# B&R Automation Studio project ABC_Pltzr (part 3)

#### paiPVSerDesMgr.typ
```iecst
(********************************************************************
 * COPYRIGHT --
 ********************************************************************
 * Package: paiFileService
 * File: paiPVSerDesMgr
 * Author: goran_2
 * Created: August 05, 2015
 ********************************************************************
 * Data types of package paiFileService
 ********************************************************************)

TYPE
	paiFSEnums_typ :
		(
		PAI_FS_PVNAME_MAXLEN := 63,
		PAI_FS_PATH_MAXLEN := 127,
		PAI_FS_TXTLEN_MID := 127,
		PAI_FS_SERDESMGR_PWRUP_NA := 0, (*PV restore option at Power Up: no action*)
		PAI_FS_SERDESMGR_PWRUP_DFLT := 1, (*PV restore option at Power Up: test storage, if different preload defaults*)
		PAI_FS_SERDESMGR_PWRUP_DFLT_fRD := 2, (*PV restore option at Power Up: test storage, if different preload defaults then read data from file*)
		PAI_FS_SERDESMGR_MAXITEMIDX := 19
		);
	paiPVSerDesChangeMonitor_typ : 	STRUCT  (*Change monitor: optional feature*)
		iChngEnable : BOOL; (*0-disabled;1-enabled*)
		iChngRejected : BOOL; (*1-reject PV changes, restore previous value*)
		iChngAccepted : BOOL; (*1-accept PV changes, store PV to file*)
		oChngDetected : BOOL; (*1-PV is changed, use information to prompt user*)
		oError : UDINT; (*1-option is enabled, but provided memory is unsufficent*)
		oState : UDINT; (*1-option is enabled, but provided memory is unsufficent*)
		iChangeMonitorMemSize : UDINT; (*size of the address space for this feature (shall be the same size or greater than the size of the PV)*)
		pChangeMonitorMem : UDINT; (*ptr to address space which has the same size as the PV (use for memory compare to detect changes)*)
	END_STRUCT;
	paiPVSerDesHMI_typ : 	STRUCT
		iBtnChangeReject : USINT;
		iBtnChangeAccept : USINT;
		iBtnSerRequest : USINT;
		iBtnDesRequest : USINT;
		oBtnVisible : USINT;
		oBtnClick : USINT;
	END_STRUCT;
	paiPVSerDesPowerUp_typ : 	STRUCT  (*Option: control of a behaivor at power up*)
		iPowerUpConfig : UDINT; (*0-nothing to do; 1-use test data; if diff, run defaults; 2-use test data; if diff, read from file*)
		iTestData : UDINT; (*Test data value (i.e. magic word 0x55555555)*)
		pTestDataStorage : UDINT; (*Ptr to the location of the magic word for this variable*)
		oError : UDINT; (*0-not ready after power up; 1-ready after power up*)
		oInitReady : UDINT; (*0-not ready after power up; 1-ready after power up*)
		oStatus : STRING[15]; (*0-not ready after power up; 1-ready after power up*)
	END_STRUCT;
	paiPVSerDesItem_typ : 	STRUCT
		iPVName : STRING[PAI_FS_PVNAME_MAXLEN]; (*PV name*)
		iDevicename : STRING[PAI_FS_PVNAME_MAXLEN]; (*Name of the file device to store PV*)
		iFilename : STRING[PAI_FS_PATH_MAXLEN]; (*Filename to store PV*)
		iSerRequest : BOOL; (*Request to write PV to file (i.e. serialize PV to file buffer > write data to  file)*)
		iDesRequest : BOOL; (*Request to read PV from file (i.e. read file to file buffer > deserialize data to PV)*)
		pPV : UDINT; (*ptr to PV*)
		iPVSize : UDINT; (*size of the PV (in bytes)*)
		pFilebuffer : UDINT; (*ptr to file r/w buffer*)
		iFilebufferSize : UDINT; (*size (bytes) of the file r/w buffer*)
		optChangeMonitor : paiPVSerDesChangeMonitor_typ; (*optional feature for automatic / HMI assisted read/write of PV-s upon changes*)
		optInitAtPowerUp : paiPVSerDesPowerUp_typ; (*optional feature: control PV init at power up; see above*)
		optPtrHMIData : REFERENCE TO paiPVSerDesHMI_typ; (*optional feature: HMI interface for PV read/write to/from file*)
		pCallbackDes : UDINT; (*deserialize callback function - processes PV deser request*)
		pCallbackSer : UDINT; (*serialize callback function - processes PV serialize request*)
		pCallbackDefault : UDINT; (*default callback function - function to set PV default values*)
		oState : UDINT; (*mgr current state*)
		oDone : UDINT; (*1 - ser or deser request is complete; *)
		oSerCount : UDINT;
		oDesCount : UDINT;
		oSerCountOld : UDINT;
		oDesCountOld : UDINT;
		oFilesizeLastSer : UDINT;
		oFilesizeLastDes : UDINT;
		oTimestampLastSer : STRING[63];
		oTimestampLastDes : STRING[63];
		oErrorCount : UDINT;
		oErrorCountOld : UDINT;
		oError : UDINT;
		oErrorTxt : STRING[PAI_FS_TXTLEN_MID];
	END_STRUCT;
	paiPVSerDesMgr_typ : 	STRUCT
		pPaiFS : UDINT;
		oState : UDINT;
		iItemCount : UDINT;
		pvItems : ARRAY[0..PAI_FS_SERDESMGR_MAXITEMIDX]OF paiPVSerDesItem_typ;
	END_STRUCT;
END_TYPE
```

#### paiFileService.var
```iecst
(********************************************************************
 * COPYRIGHT --
 ********************************************************************
 * Package: paiFileService
 * File: paiFileService.var
 * Author: goran_2
 * Created: August 05, 2011
 ********************************************************************
 * Variables of package paiFileService
 ********************************************************************)
VAR
	paiFS : paiFileService_typ := (0); (*Global PV for interfacing to PAI file service.*)
	paiFSDevices : paiFileServiceDeviceTable_typ := (0);
END_VAR
```

#### paiPVSerDesMgr.h
```c
/********************************************************************
 * COPYRIGHT --
 ********************************************************************
 * Package: paiFileService
 * File: paiPVSerDesMgr.h
 * Author: goran
 * Created: August 18, 2015
 *******************************************************************/

#include <bur/plctypes.h>

void paiPVSerDesMgrInit(paiPVSerDesMgr_typ* p);
void paiPVSerDesMgrCyclic(paiPVSerDesMgr_typ* p);

//callback functions
void paiCBWriteFileSerPV(paiFileService_typ* p, UDINT pCallbackData);
void paiCBReadFileDesPV(paiFileService_typ* p, UDINT pCallbackData);

//EOF
```

#### paiFSInterface.c
```c
/********************************************************************
 * COPYRIGHT --
 ********************************************************************
 * Package: paiFileService
 * File: paiFSInterface.c
 * Author: goran
 * Created: August 18, 2015
 *******************************************************************/

#include <bur/plctypes.h>
#ifdef _DEFAULT_INCLUDES
	#include <AsDefault.h>
#endif

#include "paiFSInterface.h"

/*
###############################################################################
Utility function to access paiFS service
###############################################################################
*/
void paiFSSetCallback(paiFileService_typ* p, UDINT pCallback, UDINT pCallbackData)
{
	if(!p)
		return;

	p->i.pCallback = pCallback;
	p->i.pCallbackData = pCallbackData;
}

void paiFSExeCallback(paiFileService_typ* p)
{
	if(!p)
		return;

	//execute fs callback to enable app to process file io
	if(p->i.pCallback){
		void (*fsCB)(paiFileService_typ* pFS, UDINT pCallbackData) =  ( void(*) (paiFileService_typ* pFS, UDINT pCallbackData) ) p->i.pCallback;
		(*fsCB)(p, p->i.pCallbackData);
	}
}

void paiFSExeCallbackCyclic(paiFileService_typ* p)
{
	//wait until request completes
	if( paiFSFileRequestIsBusy(p) )
		return;

	if( p->o.done ){
		//clear done event
		p->o.done = 0;

		//execute call back after file IO command execution is complete
		paiFSExeCallback(p);
	}
}

void paiFSDirCreateRequest(paiFileService_typ* p, UDINT adrDeviceName, UDINT adrPath, UDINT pCallback, UDINT pCallbackData)
{
	p->i.request = PAI_FS_CRDIR;
	p->i.adrName = (UDINT)adrPath;
	p->i.adrDeviceName = (UDINT) adrDeviceName;
	paiFSSetCallback(p, pCallback, pCallbackData);
}

void paiFSDirInfoRequest(paiFileService_typ* p, UDINT adrDeviceName, UDINT adrPath, UDINT pCallback, UDINT pCallbackData)
{
	p->i.request = PAI_FS_INFODIR;
	p->i.adrName = (UDINT)adrPath;
	p->i.adrDeviceName = (UDINT) adrDeviceName;
	paiFSSetCallback(p, pCallback, pCallbackData);
}

void paiFSFileDelRequest(paiFileService_typ* p, UDINT adrDeviceName, UDINT adrName, UDINT pCallback, UDINT pCallbackData)
{
	p->i.request = PAI_FS_DELFILE;
	p->i.adrName = (UDINT)adrName;
	p->i.adrDeviceName = (UDINT) adrDeviceName;
	paiFSSetCallback(p, pCallback, pCallbackData);
}

void paiFSFileRdRequest(paiFileService_typ* p, UDINT adrDeviceName, UDINT adrName, UDINT adrDst, UDINT sizeDst, UDINT pCallback, UDINT pCallbackData)
{
	p->i.request = PAI_FS_RDFILE;
	p->i.adrDeviceName = (UDINT) adrDeviceName;
	p->i.adrName = (UDINT)adrName;
	p->i.adrReadDst = (UDINT)adrDst;
	p->i.readDstLen = sizeDst;
	paiFSSetCallback(p, pCallback, pCallbackData);
}

void paiFSFileWrRequest(paiFileService_typ* p, UDINT adrDeviceName, UDINT adrName, UDINT adrSrc, UDINT sizeSrc, UDINT pCallback, UDINT pCallbackData)
{
	p->i.request= PAI_FS_WRFILE;
	p->i.adrDeviceName = (UDINT) adrDeviceName;
	p->i.adrName = (UDINT)adrName;
	p->i.adrWriteSrc = (UDINT)adrSrc;
	p->i.writeSrcLen= sizeSrc;
	paiFSSetCallback(p, pCallback, pCallbackData);
}

BOOL paiFSFileRequestIsBusy(paiFileService_typ* p)
{
	//wait until request completes
	if(p->o.busy)
		return 1;

	//reset request! IMPORTANT!
	p->i.request = PAI_FS_IDLE;
	return 0;
}

BOOL paiFSFileSystemIsInit(paiFileService_typ* p)
{
	if(!p->o.initOk)	//can't do much before paiFS completes
		return 0;

	return 1;
}
```

#### Program Logical/paiComponents/paiFileService/paiFSUnitTest

##### paiFSUnitTest.c
```c
/********************************************************************
 * COPYRIGHT --
 ********************************************************************
 * Program: paiFileTestClient
 * File: paiFileTestClient.c
 * Author: goran_2
 * Created: August 05, 2011
 ********************************************************************
 * Implementation of program paiFileTestClient
 ********************************************************************/

#include <bur/plctypes.h>

#ifdef _DEFAULT_INCLUDES
 #include <AsDefault.h>
#endif

/*
###############################################################################
PV-s
###############################################################################
*/

/*
###############################################################################
PV-s
###############################################################################
*/
#define BUF_LEN 1000
_LOCAL char txt[BUF_LEN];

_LOCAL char filename[32];

_LOCAL int readcounterok ;
_LOCAL int readcountererr ;

_LOCAL int writecounterok ;
_LOCAL int writecountererr ;

_LOCAL int myInitDone;

/*
###############################################################################
Init, Cyclic, Exit
###############################################################################
*/
void _INIT paiFileTestClientINIT( void )
{
	/* TODO: Add code here */
	myInitDone = 0;
}

void _CYCLIC paiFileTestClientCYCLIC( void )
{
	/* TODO: Add code here */

	/*wait till file service ready then init application access to file service*/
	if(!myInitDone && paiFS.io.initOk){
		myInitDone = 1;
		/*copy filename into a buffer so it may be changed from the watch window*/
		strcpy(filename, "appcfg.txt");
		paiFS.io.fileName = (UDINT)filename;

		/*in this example same buffer used for read and write*/
		paiFS.io.readDstAdr = (UDINT)txt;
		paiFS.io.readDstLen = BUF_LEN;
		paiFS.io.writeSrcAdr= (UDINT)txt;

		/*aux PV-s to monitor the activity*/
		readcounterok = 0;
		readcountererr = 0;

		writecounterok = 0;
		writecountererr = 0;
	}

	/*in this example continously update length for write request. That way, when writeRequest get's issued from watch window, correct value gets set!*/
	paiFS.io.writeSrcLen = strlen(&txt[0]);

	/*example on how to monitor if file service has completed a request*/
	if(paiFS.io.readDone){
		/*reset signal here*/
		paiFS.io.readDone = 0;

		if(paiFS.io.status)
			readcountererr++;
		else
			readcounterok++;
	}

	if(paiFS.io.writeDone){
		/*reset signal here*/
		paiFS.io.writeDone = 0;

		if(paiFS.io.status)
			writecountererr++;
		else
			writecounterok++;
	}
}

void _EXIT paiFileTestClientEXIT( void )
{
	/* TODO: Add code here */
}
```

### Program Logical/paiComponents/paiHmi

#### paiHmiCmd.typ
```iecst
(********************************************************************
 * COPYRIGHT -- pai
 ********************************************************************
 * Package: HMI
 * File: HMI.typ
 * Author: goran
 * Created: August 28, 2013
 ********************************************************************
 * Data types of package HMI
 ********************************************************************)
(*==========================*)
(*==== HMI Command Interface ==*)
(*==========================*)

TYPE
	hmiCmd_typ : 	STRUCT
		main : hmiCmdMain_typ;
		infeed : hmiCmdInfeed_typ;
		outfeed : hmiCmdOutfeed_typ;
		qc : hmiCmdQC_typ;
		lights : hmiCmdLights_typ;
		diag : hmiCmdDiag_typ;
		listQCInspectors : STRING[511];
	END_STRUCT;
	hmiCmdX20Outfeed_typ : 	STRUCT  (*command to control / force an OUTFEED output module*)
		doDoorWeigh : BOOL; (*weigh door*)
		doBelt : BOOL; (*belt control clutch*)
		doQC1 : BOOL; (*qc1 diverter *)
		doQC2 : BOOL; (*qc2 diverter*)
	END_STRUCT;
	hmiCmdX20Station_typ : 	STRUCT  (*command to control / force an STATION output module(s)*)
		doTakeout0 : BOOL; (*takeout (0 + moduleNum*4)*)
		doTakeout1 : BOOL; (*takeout (1 + moduleNum*4)*)
		doTakeout2 : BOOL; (*takeout (2 + moduleNum*4)*)
		doTakeout3 : BOOL; (*takeout (3 + moduleNum*4)*)
		doDumpAll : BOOL; (*station dump ALL (0..3 + moduleNum*4)*)
		doDump0 : BOOL; (*station dump (0 + moduleNum*4)*)
		doDump1 : BOOL; (*station dump (1 + moduleNum*4)*)
		doDump2 : BOOL; (*station dump (2 + moduleNum*4)*)
		doDump3 : BOOL; (*station dump (3 + moduleNum*4)*)
		doLights : BOOL; (*state of outputs (bit map)*)
	END_STRUCT;
	hmiCmdX20Infeed_typ : 	STRUCT  (*command to control / force an INFEED output module*)
		doDoorBuffer : BOOL; (*buffer door*)
		doDoorWeigh : BOOL; (*weigh door*)
		doLine : BOOL; (*line control valve*)
	END_STRUCT;
	hmiCmdIO_typ : 	STRUCT  (*command to control/force outputs of the entire machine*)
		enableDOForce : UDINT; (*enable DO force *)
		infeed : hmiCmdX20Infeed_typ; (*infeed*)
		outfeed : hmiCmdX20Outfeed_typ; (*outfeed*)
		stations : ARRAY[0..30]OF hmiCmdX20Station_typ; (*stations*)
	END_STRUCT;
	hmiCmdLights_typ : 	STRUCT
		enableLightControl : UDINT; (*0-Lights control feature off; 1-Lights control feature on; 2-Lights control test mode*)
		LightsDO : ARRAY[0..30]OF UDINT; (*Bit mapped Light outputs; A UDINT per station*)
	END_STRUCT;
	hmiCmdInfeed_typ : 	STRUCT
		scaleCalibration : hmiCmdScaleCalib_typ;
		pauseOperation : UDINT; (*0-normal 1-pause operation*)
		gateEnable : UDINT; (*gate enable bit array (bit encoded UDINT), bit0-station 1*)
	END_STRUCT;
	hmiCmdDiag_typ : 	STRUCT
		alarmsAck : ARRAY[0..19]OF UDINT;
		io : hmiCmdIO_typ; (*control of the outputs from the Windows side (testing and troubleshooting)*)
	END_STRUCT;
	hmiCmdScaleCalib_typ : 	STRUCT
		calibrationCmd : UDINT; (*Calibration command: 0-normal operation;1-doZero;2-doCalibration*)
		calibrationWt : REAL; (*Calibraton wt*)
	END_STRUCT;
	hmiCmdX20DO_typ : 	STRUCT  (*command to control / force an X20 DO output module*)
		out : UDINT; (*state of outputs (bit map)*)
	END_STRUCT;
	hmiCmdQC_typ : 	STRUCT
		stationQCEnabled : UDINT; (*bit codded UDINT indicating a station for QC (bit0-station1, etc)*)
		QCMode : UDINT; (*0-stop the outfeed if needed to wait for QC; 1-don't stop the outfeed even if QC is needed for the current station (i.e. never stop the outfeed to wait for QC to complete)*)
		workerScoreAtQC : UDINT; (*score of the worker that is currently inspected at QC (uses status.qc.stationInQC)*)
		workerNameAtQC : STRING[31]; (*name of the worker that is currently inspected at QC (uses status.qc.stationInQC)*)
		workerScoreAtQC2 : UDINT; (*score of the worker that is currently inspected at QC2 (uses status.qc.stationInQC2)*)
		workerNameAtQC2 : STRING[31]; (*name of the worker that is currently inspected at QC2 (uses status.qc.stationInQC2)*)
	END_STRUCT;
	hmiCmdMain_typ : 	STRUCT
		machineState : UDINT; (*0-stopped;1-filling;2-run;3-washdown*)
	END_STRUCT;
	hmiCmdOutfeed_typ : 	STRUCT
		scaleCalibration : hmiCmdScaleCalib_typ;
		pauseOperation : UDINT; (*0-normal 1-pause operation*)
	END_STRUCT;
END_TYPE
```

#### paiHmiDropdwMenuRT.typ
```iecst
(********************************************************************
 * COPYRIGHT -- pai
 ********************************************************************
 * Package: HMI
 * File: HMI.typ
 * Author: goran
 * Created: August 28, 2013
 ********************************************************************
 * Data types of package HMI
 ********************************************************************)
(*########################################################################*)
(*HMI object - Dropdown Menu located at the Upper Right side of the screen*)
(*########################################################################*)

TYPE
	paiHmiDropdownMenuRTEnums_typ :
		(
		paiHMI_ENUM_MENU_ITEMS_RT := 10 (*Main menu - right side - number of buttons*)
		);
	paiHmiDropdwMenuRT_typ : 	STRUCT
		iMenuIndexRT : INT;
		iMenuRTTimeout : REAL; (*Duration after which a dropdown menu is automaticaly hiden if not clicked *)
		oMenuIndexRT : INT; (*Main menu currently selected menu item - RT*)
		oMenuVisible : INT;
		oMenuVisibleItems : ARRAY[0..paiHMI_ENUM_MENU_ITEMS_RT]OF INT; (*1-items is not visible*)
		oMenuDisabledItems : ARRAY[0..paiHMI_ENUM_MENU_ITEMS_RT]OF BOOL; (*1-Item is disabled*)
		iMenuSelectItem : ARRAY[0..paiHMI_ENUM_MENU_ITEMS_RT]OF BOOL; (*an input array to select items from the code; first found 1 will be selected;*)
		oMenuSelectedItems : ARRAY[0..paiHMI_ENUM_MENU_ITEMS_RT]OF BOOL; (*1-Item is currently selected (indexRT)*)
		oMenuPressedItems : ARRAY[0..paiHMI_ENUM_MENU_ITEMS_RT]OF BOOL; (*1-an item that was pressed, single shot*)
		mMenuVisibleOld : INT;
		menuRTHideTimer : TON;
	END_STRUCT;
END_TYPE
```

#### paiHmiMsgRunning.typ
```iecst
(********************************************************************
 * COPYRIGHT -- pai
 ********************************************************************
 * Package: HMI
 * File: HMI.typ
 * Author: goran
 * Created: August 28, 2015
 ********************************************************************
 * Data types of package HMI
 ********************************************************************)
(*########################################################################*)
(*HMI object - Running Messages (i.e. content scrolls )*)
(*########################################################################*)

TYPE
	paiHmiMsgRunningEnum_typ :
		(
		paiHMI_ENUM_RUNMSG_MAXLEN := 255 (*Main menu - left side - number of buttons*)
		);
	paiHmiMsgRunning_typ : 	STRUCT  (*0-disable; 1-enable*)
		iEnable : BOOL; (*input: address of the alarm array*)
		iScrollMode : UDINT; (*scroll mode*)
		iScrollLength : UDINT; (*scroll length*)
		iScrollDelayXms : UDINT; (*scroll speed*)
		iMsgAddr : UDINT; (*address of the message for scroll*)
		oMsg : STRING[255]; (*output: message ID of the active alarm / message*)
		oMsgVisible : UINT; (*output: visibilty control DP for the VC text message*)
		oMsgFCIdx : UINT; (*output: visibilty control DP for the VC text message*)
		state : UINT; (*Status for common dialog layer*)
		curIdx : UINT; (*Status for common dialog layer*)
		tmr1 : TON; (*Dialog control timer*)
	END_STRUCT;
END_TYPE
```

#### paiHMIParamListTable.typ
```iecst
(********************************************************************
 * COPYRIGHT -- pai
 ********************************************************************
 * Package: HMI
 * File: HMI.typ
 * Author: goran
 * Created: August 28, 2013
 ********************************************************************
 * Data types of package HMI
 ********************************************************************)

TYPE
	hmiParamListEnums_typ :
		(
		hmiTableMAXENUMS := 10, (*Max number of items in an enum list when property type is enum*)
		hmiTableMAXENUMTEXT := 15, (*Max len of each enum text*)
		hmiTableMAXENTRIES := 50, (*Max number of supported properties in the property list*)
		hmiTableMAXDESCRIPTION := 255, (*Max length of the description text for each property*)
		hmiTableMAXNAME := 31 (*Max name of a property*)
		);
END_TYPE

(*########################################################################*)
(*HMI object - PARAMETER LIST - LIMITS*)
(*########################################################################*)

TYPE
	hmiParamLimits_typ : 	STRUCT
		k_factor : REAL; (*scaling k factor (y=kx + n, where y=dsiplay value, x=plc value)*)
		n_factor : REAL; (*scaling n factor (y=kx + n, where y=dsiplay value, x=plc value)*)
		minValue : REAL; (*min value*)
		maxValue : REAL; (*max value*)
		defaultValue : REAL; (*default value*)
		pEnumText : UDINT; (*ptr to a string of comma delimited enum texts*)
		pEnumVals : UDINT; (*ptr to a string of comma delimited enum values*)
		valueType : UINT; (*type of the paramvalue (0-DINT, 1-REAL, 2-ENUM)*)
	END_STRUCT;
END_TYPE

(*########################################################################*)
(*HMI object - PARAMETER LIST*)
(*########################################################################*)

TYPE
	hmiParamListTable_typ : 	STRUCT
		listHeader : STRING[hmiTableMAXNAME]; (*name of the list (header text)*)
		listIdText : ARRAY[0..hmiTableMAXENTRIES]OF STRING[7]; (*table colum: id-s*)
		listValueText : ARRAY[0..hmiTableMAXENTRIES]OF STRING[15]; (*table colum: value*)
		listName : ARRAY[0..hmiTableMAXENTRIES]OF STRING[hmiTableMAXNAME]; (*table colum: name*)
		listDescription : ARRAY[0..hmiTableMAXENTRIES]OF STRING[hmiTableMAXDESCRIPTION]; (*table colum: description*)
		listValuePtr : ARRAY[0..hmiTableMAXENTRIES]OF UDINT; (*list of ptrs to parametars*)
		listDecPlaces : ARRAY[0..hmiTableMAXENTRIES]OF DINT; (*list of dec places for each parametar*)
		listLimits : ARRAY[0..hmiTableMAXENTRIES]OF hmiParamLimits_typ;
		selName : STRING[hmiTableMAXNAME]; (*name of the currently selected/active parametar*)
		selDescription : STRING[hmiTableMAXDESCRIPTION]; (*description of the currently selected/active parametar*)
		listSelValueEnumText : ARRAY[0..hmiTableMAXENUMS]OF STRING[hmiTableMAXENUMTEXT]; (*list of available enum text for a property that is of type ENUM*)
		listSelValueEnum : ARRAY[0..hmiTableMAXENUMS]OF UDINT; (*list of available enum text for a property that is of type ENUM*)
		selValueEnumIndex : UDINT; (*value of the currently selected/active parametar for type enum*)
		selValueEnumIndexMax : UDINT; (*value of the currently selected/active parametar for type enum*)
		selValueREAL : REAL; (*value of the currently selected/active parametar*)
		selValueREALOld : REAL; (*value of the currently selected/active parametar (previous value for change detection*)
		selValueREALMax : REAL; (*max value of the currently selected/active parametar*)
		selValueREALMin : REAL; (*min value of the currently selected/active parametar*)
		selValueREALDefault : REAL; (*default value of the currently selected/active parametar*)
		selValueDecPlaces : DINT; (*default value of the currently selected/active parametar*)
		selValueDINT : DINT; (*value of the currently selected/active parametar*)
		selValueDINTOld : DINT; (*value of the currently selected/active parametar (previous value for change detection*)
		selValueDINTMax : DINT; (*max value of the currently selected/active parametar*)
		selValueDINTMin : DINT; (*min value of the currently selected/active parametar*)
		selValueDINTDefault : DINT; (*default value of the currently selected/active parametar*)
		selValueFormVisible : DINT; (*visibility control of the form / controls for setting parametar value*)
		index : UINT; (*index of the currently selected/active parametar*)
		indexOld : UINT; (*index of the currently selected/active parametar (previous value for change detection)*)
		maxIndex : UINT; (*max index / number of items in the table. Must be less then hmiTableMAXDESCRIPTION!!!*)
		setDefaultRequest : BOOL; (*set default request flag*)
	END_STRUCT;
END_TYPE
```

#### paiHmiStatus.typ
```iecst
(********************************************************************
 * COPYRIGHT -- pai
 ********************************************************************
 * Package: HMI
 * File: HMI.typ
 * Author: goran
 * Created: August 28, 2013
 ********************************************************************
 * Data types of package HMI
 ********************************************************************)
(*########################################################################*)
(*HMI object - Status message (data from real-time to HMI)*)
(*########################################################################*)

TYPE
	hmiStatus_typ : 	STRUCT
		main : hmiStatusMain_typ;
		infeed : hmiStatusInfeed_typ;
		outfeed : hmiStatusOutfeed_typ;
		qc : hmiStatusQC_typ;
		lights : hmiStatusLights_typ;
		diag : hmiStatusDiag_typ;
	END_STRUCT;
	hmiStatusOutfeed_typ : 	STRUCT
		wt : REAL; (*current outfeed wt *)
		status : UDINT; (*current state of the outfeed subsystem*)
		zeroTabCounter : UDINT; (*increments each time a zeroTab gets detected. Reset to 0 after power up.*)
	END_STRUCT;
	hmiStatusInfeed_typ : 	STRUCT
		wt : REAL; (*current infeed wt *)
		state : UDINT; (*current state of the infeed subsystem*)
	END_STRUCT;
	hmiStatusIOInfeed_typ : 	STRUCT  (*infeed IO*)
		x2xBuxRx : hmiStatusX20TR_typ; (*x2x bus rx module*)
		wt : hmiStatusX20AI_typ; (*wt analog input*)
		DOModule : hmiStatusX20DO_typ; (*infeed outputs*)
		x2xBuxTx : hmiStatusX20TR_typ; (*x2x bus tx module*)
	END_STRUCT;
	hmiStatusDiag_typ : 	STRUCT
		state : UDINT; (*current state of the Diag subsystem*)
		alarms : ARRAY[0..19]OF UDINT;
		io : hmiStatusIO_typ; (*status of IO for display on the windows side*)
		dummy : UDINT;
	END_STRUCT;
	hmiStatusLights_typ : 	STRUCT
		dummy : UDINT;
	END_STRUCT;
	hmiStatusMain_typ : 	STRUCT
		state : UDINT; (*current state of the main subsystem*)
	END_STRUCT;
	hmiStatusIO_typ : 	STRUCT  (*status of the entire machine IO*)
		infeed : hmiStatusIOInfeed_typ; (*infeed*)
		outfeed : hmiStatusIOOutfeed_typ; (*outfeed*)
		stations : ARRAY[0..30]OF hmiStatusIOStation_typ; (*stations*)
	END_STRUCT;
	hmiStatusIOOutfeed_typ : 	STRUCT  (*infeed IO*)
		x2xBuxRx : hmiStatusX20TR_typ; (*x2x bus rx module*)
		wt : hmiStatusX20AI_typ; (*wt analog input*)
		DIModule : hmiStatusX20DI_typ; (*infeed inputs*)
		DOModule : hmiStatusX20DO_typ; (*outfeed outputs*)
		x2xBuxTx : hmiStatusX20TR_typ; (*x2x bus tx module*)
	END_STRUCT;
	hmiStatusIOStation_typ : 	STRUCT  (*infeed IO*)
		x2xBuxRx : hmiStatusX20TR_typ; (*x2x bus rx module*)
		DIModule : hmiStatusX20DI_typ; (*station inputs*)
		DOLights : hmiStatusX20DO_typ; (*station light outputs*)
		DOModule : hmiStatusX20DO_typ; (*station outputs*)
		x2xBuxTx : hmiStatusX20TR_typ; (*x2x bus tx module*)
	END_STRUCT;
	hmiStatusX20DO_typ : 	STRUCT  (*status of an X20 DO output module*)
		moduleOk : UDINT; (*moduleOk bit map (only bit0 used)*)
		out : UDINT; (*state of outputs (bit map)*)
		outStatus : UDINT; (*status of outputs (bit map)*)
	END_STRUCT;
	hmiStatusX20TR_typ : 	STRUCT  (*status of an X20 bus Tx or bus Rx  module*)
		moduleOk : UDINT; (*moduleOk bit map (only bit0 used)*)
		statusInput01 : UDINT; (*see module description (bit map, only bit 0 used)*)
		statusInput02 : UDINT; (*see module description (bit map, only bit 0 used)*)
	END_STRUCT;
END_TYPE

(*==========================*)
(*==== IO Status Support      ====*)
(*==========================*)

TYPE
	hmiStatusX20DI_typ : 	STRUCT  (*status of an X20 DI input module*)
		moduleOk : UDINT; (*moduleOk bit map (only bit0 used)*)
		in : UDINT; (*state of inputs (bit map)*)
		notused : UDINT; (*state of inputs (bit map)*)
	END_STRUCT;
	hmiStatusQC_typ : 	STRUCT
		state : UDINT; (*current state of the QC subsystem*)
		stationInQC : UDINT; (*number of the station beeing currently inspected at the QC*)
		stationInQC2 : UDINT; (*number of the station beeing currently inspected at the QC2*)
	END_STRUCT;
	hmiStatusX20AI_typ : 	STRUCT  (*status of an X20 DO output module*)
		moduleOk : UDINT; (*moduleOk bit map (only bit0 used)*)
		inAnalog : DINT; (*analog input value*)
		inStatus : UDINT; (*analog input status*)
		config : UDINT; (*analog input configuraton*)
	END_STRUCT;
END_TYPE
```

#### paiHmiDialog.h
```c
/********************************************************************
 * COPYRIGHT -- pai
 ********************************************************************
 * Program: hmilogic
 * File: hmiDialog.h
 * Author: goran
 * Created: September 05, 2013
 *******************************************************************/

#include <bur/plctypes.h>
#ifdef _DEFAULT_INCLUDES
#include <AsDefault.h>
#endif
BOOL paiHmiDialogIsActive(paiHmiDialog_typ* p);
void paiHmiDialogHide(paiHmiDialog_typ* p);
void paiHmiDialogShow(paiHmiDialog_typ* p, char* msg, UINT timeout_ms, UINT resultForOk, UINT resultForCancel, UINT timeoutConfig);
UINT paiHmiDialogCyclic(paiHmiDialog_typ* p);
```

#### paiHmiMsgScrolling.h
```c
/********************************************************************
 * COPYRIGHT --
 ********************************************************************
 * Package: paiHmiTemplate
 * File: paiHmiMsgScrolling.h
 * Author: goran
 * Created: July 29, 2015
 *******************************************************************/

#include <bur/plctypes.h>
#ifdef _DEFAULT_INCLUDES
	#include <AsDefault.h>
#endif
void paiHmiMsgScrollingInit(paiHmiMsgScrolling_typ* p, UDINT pAlarmArray, UDINT alarmArrayLen, UDINT msgTimeXms);
void paiHmiMsgScrollingCyclic(paiHmiMsgScrolling_typ* p);
```

#### paiHmiParamList.h
```c
/********************************************************************
 * COPYRIGHT -- pai
 ********************************************************************
 * Program: hmilogic
 * File: hmiParamList.h
 * Author: goran
 * Created: September 05, 2013
 *******************************************************************/
#include <bur/plctypes.h>
#ifdef _DEFAULT_INCLUDES
#include <AsDefault.h>
#endif
void hmiParamListTableCyclic(hmiParamListTable_typ* p);
void hmiParamListTableEntryLast(hmiParamListTable_typ* p);
void hmiParamListTableEntryFirst(hmiParamListTable_typ* p, char* pListName);
 void hmiParamListTableAddEntryNext(hmiParamListTable_typ* p, UDINT pValue, char* pName, REAL valDefault, REAL valMin, REAL valMax, int decPlaces, REAL k_factor, REAL n_factor, UINT valueType, char* pDescription);
```

#### paiHmiSystemNetworking.h
```c
/********************************************************************
 * COPYRIGHT -- pai
 ********************************************************************
 * Program: hmilogic
 * File: hmiAlert.h
 * Author: goran
 * Created: September 05, 2013
 *******************************************************************/

#include <bur/plctypes.h>
#ifdef _DEFAULT_INCLUDES
#include <AsDefault.h>
#endif
void paiHmiSystemNetworkingInit(paiHmiSystemNetworking_typ* p);
void paiHmiSystemNetworkingCyclic(paiHmiSystemNetworking_typ* p);
```

#### paiHmiDropdownMenuRT.c
```c
/********************************************************************
 * COPYRIGHT --
 ********************************************************************
 * Package: paiHmiTemplate
 * File: paiHmiDropdownMenuRT.c
 * Author: goran
 * Created: July 29, 2015
 *******************************************************************/

#include <bur/plctypes.h>
#ifdef _DEFAULT_INCLUDES
	#include <AsDefault.h>
#endif

//logic control of the global MENU KEYS on the Left Side (i.e. STOPPED, FILLING, PRODUCTION, ...)
void paiHmiDropDownMenuRTInit(paiHmiDropdwMenuRT_typ* p)
{
	//menu not visible at start
	p->oMenuVisible = 1;
}

//logic control of the global MENU KEYS on the Left Side (i.e. STOPPED, FILLING, PRODUCTION, ...)
void paiHmiDropDownMenuRTCyclic(paiHmiDropdwMenuRT_typ *p)
{
	int ii;

	//process input array to allow selection of menu items from the program
	for(ii=0; ii<=paiHMI_ENUM_MENU_ITEMS_RT;ii++){
		if(p->iMenuSelectItem[ii]){
			p->iMenuSelectItem[ii] = 0;
			p->iMenuIndexRT = ii;
			break;
		}
	}

	//set a bit within an array of the item that is currently selected
	for(ii=0; ii<=paiHMI_ENUM_MENU_ITEMS_RT;ii++){
		p->oMenuSelectedItems[ii] = 0;
		if(ii == p->iMenuIndexRT){
			p->oMenuSelectedItems[ii] = 1;
		}
	}

	bgTimerCyclic(&p->menuRTHideTimer);

	//clear all single shot flags
	for(ii=0; ii<=paiHMI_ENUM_MENU_ITEMS_RT;ii++){
		p->oMenuPressedItems[ii] = 0;
	}
	//generate single shot for a button press
	if(p->oMenuIndexRT != p->iMenuIndexRT){
		p->oMenuPressedItems[p->iMenuIndexRT] = 1;
	}
	p->oMenuIndexRT = p->iMenuIndexRT;

	//when menu becomes visible > start the timer
	if(!p->oMenuVisible && p->mMenuVisibleOld){
		bgTimerStart(&p->menuRTHideTimer, p->iMenuRTTimeout * 1000); //dropdown timer LF
	}
	p->mMenuVisibleOld = p->oMenuVisible;
	//if menu still visible after timer expires > hide menu
	if( !p->oMenuVisible && bgTimerIsTimeOut(&p->menuRTHideTimer) ){
		p->oMenuVisible = 1;
	}

}
```

#### paiHmiLFMenuTabsPages.c
```c
/********************************************************************
 * COPYRIGHT --
 ********************************************************************
 * Package: paiHmiTemplate
 * File: paiHmiTemplateLogic.c
 * Author: goran
 * Created: July 27, 2015
 *******************************************************************/

#include <bur/plctypes.h>
#ifdef _DEFAULT_INCLUDES
	#include <AsDefault.h>
#endif

#include "../bglib/bgstring.h"

#define paiHMI_KEYWORD_COMMENT "//"
#define paiHMI_KEYWORD_BUTTON "BUTTON:"
#define paiHMI_KEYWORD_TAB "TAB:"
#define paiHMI_KEYWORD_DELIM ","

//copy current tab setting to current tab PV-s
static void menuTabSetCurrent(paiHmiTemplate_typ* p, int tabIndex){
	if(!p)
		return;

	brsmemcpy((UDINT)p->activeTabs, (UDINT)p->prv.menuLF[p->currentMenuLF].tabs , sizeof(p->activeTabs));

	//activate first tab
	p->keys.tabKeysRadioDataPoint = tabIndex;
}

static void menuTopLFSetCurrent(paiHmiTemplate_typ* p){
	if(!p)
		return;

	brsmemcpy((UDINT)&p->activeTopMenuLF, (UDINT)&p->prv.menuLF[p->currentMenuLF].button , sizeof(p->activeTopMenuLF));
}

//logic control of the tab key operation (i.e. radio button fuction)
static void menuButtonsVisibility(paiHmiTemplate_typ* p, int visible)
{
int ii;

	for(ii = 0; ii<paiHMI_ENUM_MENU_ITEMS_LT; ii++){
		if(!p->prv.menuLF[ii].button.itemDisabled){
			p->prv.menuLF[ii].button.itemVisible = visible;
		}else{
			p->prv.menuLF[ii].button.itemVisible = 1;//not visible
		}
	}
}

static void menuPageChange(paiHmiTemplate_typ* p, UINT newPage)
{
	//activate first tab (applies to any screen)
	p->runtime.pageChange = newPage;
	p->prv.pageSetByLFMenu = newPage;
}

static void menuCyclicTabKeys(paiHmiTemplate_typ* p);

//logic control of the global MENU KEYS on the Left Side
static void menuCyclicKeysLF(paiHmiTemplate_typ* p)
{
	static int menuVisibleLTOld = 0;

	bgTimerCyclic(&p->status.menuLFHideTimer);

	//top button pressed?
	if(p->keys.menuKeyTopLT){
		p->keys.menuKeyTopLT = 0;
		if(p->status.menuVisibleLT){
			p->status.menuVisibleLT = 0;
		}else{
			p->status.menuVisibleLT = 1;
		}
	}

	//menu item pressed?
	if((p->keys.currentMenuLF >= 0) && (p->keys.currentMenuLF <= paiHMI_ENUM_MENU_ITEMS_LT)){
		p->currentMenuLF = p->keys.currentMenuLF;
		p->keys.currentMenuLF = -1;
		menuPageChange(p, p->prv.menuLF[p->currentMenuLF].button.jumpPageId);
		p->status.menuVisibleLT = 1;
		menuTopLFSetCurrent(p);
		//if(p->keys.tabKeysRadioDataPoint){
		//	p->keys.tabKeysRadioDataPointOld = 0;
		//	brsmemcpy((UDINT)p->activeTabs, (UDINT)p->prv.menuLF[p->currentMenuLF].tabs , sizeof(p->activeTabs));
		//	menuCyclicTabKeys(p);
		//}else{
			menuTabSetCurrent(p, 1);
		//}
	}

	//when menu becomes visible > start the timer
	if(!p->status.menuVisibleLT && menuVisibleLTOld){
		bgTimerStart(&p->status.menuLFHideTimer, 5000); //dropdown timer LF
		menuButtonsVisibility(p, 0);//show menu items
	}

	if(p->status.menuVisibleLT && !menuVisibleLTOld){
		menuButtonsVisibility(p, 1);//hide menu items
	}

	menuVisibleLTOld = p->status.menuVisibleLT;
	//if menu still visible after timer expires > hide menu
	if( !p->status.menuVisibleLT && bgTimerIsTimeOut(&p->status.menuLFHideTimer) ){
		p->status.menuVisibleLT = 1;
	}

}

//logic control of the tab key operation (i.e. radio button function)
static void menuCyclicTabKeys(paiHmiTemplate_typ* p)
{
	int ii;
	for(ii=0;ii<=paiHMI_ENUM_TABS_MAXIDX;ii++){

		if(p->keys.tabKeysRadioDataPoint != p->keys.tabKeysRadioDataPointOld){
			p->keys.tabKeysRadioDataPointOld = p->keys.tabKeysRadioDataPoint;
			menuPageChange(p, p->activeTabs[p->keys.tabKeysRadioDataPoint].jumpPageId );
		}

		if(ii == p->keys.tabKeysRadioDataPoint){
			p->keys.tabKeysRadioArray[ii] = 1;//select array elements that matches selected radio button
		}else{
			p->keys.tabKeysRadioArray[ii] = 0;//unselect all other array elements
		}
	}
}

static void paiHmiDefineTab(paiHmiTemplate_typ* p){
int offset;
int keywordLen;
char* pItemLine;
char *pItemTextEnd;
char *pItemPageNum;

	if(!p || !p->prv.indexButton)
		return;

	//Process following line (example):
	//    +------------------ keyword
	//    |     +------------ item label
	//    |     |     +------ page index for jump
	//    |     |     |
	//"TAB: Main, 10
	keywordLen = brsstrlen((UDINT)paiHMI_KEYWORD_TAB);
	offset = bgStrFind(p->prv.text, paiHMI_KEYWORD_TAB, 0, keywordLen);
	pItemLine = &p->prv.text[offset + keywordLen];

	//find 1st comma
	keywordLen = brsstrlen((UDINT)paiHMI_KEYWORD_DELIM);
	offset = bgStrFind(pItemLine, paiHMI_KEYWORD_DELIM, -1, -1);
	if(offset < 0){
		return;
	}
	pItemTextEnd = &pItemLine[offset];
	pItemPageNum = pItemTextEnd + keywordLen;

	//copy item label text
	brsmemcpy((UDINT)p->prv.menuLF[p->prv.indexButton - 1].tabs[p->prv.indexTab].itemText, (UDINT)pItemLine, pItemTextEnd - pItemLine);
	p->prv.menuLF[p->prv.indexButton - 1].tabs[p->prv.indexTab].itemText[offset] = 0;

	//get jumpPageIdx
	p->prv.menuLF[p->prv.indexButton - 1].tabs[p->prv.indexTab].jumpPageId = brsatoi((UDINT)pItemPageNum);
	p->prv.menuLF[p->prv.indexButton - 1].tabs[p->prv.indexTab].itemVisible = 0;//visible
	p->prv.menuLF[p->prv.indexButton - 1].tabs[p->prv.indexTab].itemDisabled = 0;//not disabled

	//increment button index; reset tab index
	p->prv.indexTab++;
}

static void paiHmiDefineButton(paiHmiTemplate_typ* p){
int offset;
int keywordLen;
char* pItemLine;
char *pItemTextEnd;
char *pItemPageNum;

	if(!p)
		return;

	//Process following line (example):
	//    +------------------ keyword
	//    |     +------------ item label
	//    |     |     +------ page index for jump
	//    |     |     |
	//"BUTTON: Main, 10
	keywordLen = brsstrlen((UDINT)paiHMI_KEYWORD_BUTTON);
	offset = bgStrFind(p->prv.text, paiHMI_KEYWORD_BUTTON, 0, keywordLen);
	pItemLine = &p->prv.text[offset + keywordLen];

	//find 1 comma
	keywordLen = brsstrlen((UDINT)paiHMI_KEYWORD_DELIM);
	offset = bgStrFind(pItemLine, paiHMI_KEYWORD_DELIM, -1, -1);
	if(offset < 0){
		return;
	}
	pItemTextEnd = &pItemLine[offset];
	pItemPageNum = pItemTextEnd + keywordLen;

	//copy text
	brsmemcpy((UDINT)p->prv.menuLF[p->prv.indexButton].button.itemText, (UDINT)pItemLine, pItemTextEnd - pItemLine);
	p->prv.menuLF[p->prv.indexButton].button.itemText[offset] = 0;

	//get jumpPageIdx
	p->prv.menuLF[p->prv.indexButton].button.jumpPageId = brsatoi((UDINT)pItemPageNum);
	p->prv.menuLF[p->prv.indexButton].button.itemDisabled = 0;//not disabled

}

static void paiHmiDefinePageNavigation(paiHmiTemplate_typ* p){
int ii;
int jj;

	if(!p)
		return;

	//clear parsing error
	brsstrcpy((UDINT)p->prv.parseErrorText, (UDINT)"");

	//make all buttons and tabs NOT VISIBLE
	for(jj=0; jj <= paiHMI_ENUM_MENU_ITEMS_LT; jj++){
		p->prv.menuLF[jj].button.itemVisible = 1;//not visible
		p->prv.menuLF[jj].button.itemDisabled = 1;//disabled
		for(ii = 0; ii <= paiHMI_ENUM_TABS_MAXIDX ; ii++){
			p->prv.menuLF[jj].tabs[ii].itemVisible = 1;//not visible
		}
	}

	//reset tab / button indexes
	p->prv.indexTab = 1;//Start from index 1; Index 0 not used!
	p->prv.indexButton = 0;

	for(p->prv.index = 0; p->prv.index <= paiHMI_ENUM_TG_TEXT_MAXIDX; p->prv.index++ ){

		bgStrCpyN(p->prv.text, p->prv.textLines[p->prv.index], sizeof(p->prv.text));

		if( bgStrFind(p->prv.text, paiHMI_KEYWORD_COMMENT, 0, brsstrlen((UDINT)paiHMI_KEYWORD_COMMENT)) >= 0){
			//comment: skip this line
			continue;
		}

		if( bgStrFind(p->prv.text, paiHMI_KEYWORD_BUTTON, 0, brsstrlen((UDINT)paiHMI_KEYWORD_BUTTON))  >= 0 ){
			//button: process button line
			paiHmiDefineButton(p);
			//increment button index; reset tab index
			p->prv.indexButton++;
			p->prv.indexTab = 1;
			continue;
		}

		if( bgStrFind(p->prv.text, paiHMI_KEYWORD_TAB, 0, brsstrlen((UDINT)paiHMI_KEYWORD_TAB)) >= 0 ){
			//tab: process tab line
			paiHmiDefineTab(p);
			continue;
		}
	}

}

static void paiHmiIncTxtIndex(paiHmiTemplate_typ* p){
	if(!p)
		return;

	p->prv.index++;
	if(p->prv.index > paiHMI_ENUM_TG_TEXT_MAXIDX ){
		 p->prv.state = 3;
	}
}

static void paiHmiGetTGText(paiHmiTemplate_typ* p){
	if(!p)
		return;
	brsstrcpy((UDINT)p->prv.textLines[p->prv.index], (UDINT)&p->prv.text);
}

/** Tabs logic */
static void paiHmiParsePageNavigationTG(paiHmiTemplate_typ* p, char* pVisuName, UDINT indexOfTGForHmiNavigation){
	UINT status;

	if(!p || !pVisuName || p->prv.initDone)
		return;

	switch(p->prv.state){
		case 0:
			p->prv.vcHandle = VA_Setup(1 , pVisuName);
			if(p->prv.vcHandle){
				p->prv.state = 1;
				p->prv.index = 0;
			}
		break;
		case 1:
	   		if( VA_Saccess(1, p->prv.vcHandle) )
				return;

			p->prv.textLen = sizeof(p->prv.text);
	        status = VA_GetTextByTextGroup(1, p->prv.vcHandle, indexOfTGForHmiNavigation, p->prv.index, (UDINT)p->prv.text,(UDINT)&p->prv.textLen);
			if(!status){
			 	//Text read ok; get next text
				paiHmiGetTGText(p);
				paiHmiIncTxtIndex(p);
			}else
			if(status == vaERR_BUSY){

			}else
			if(status == vaERR_PARAMETER){
				paiHmiIncTxtIndex(p);
			}else{
				p->prv.state = 2;
			}
	        VA_Srelease(1, p->prv.vcHandle);
		break;
		case 2:
		//error state
		break;
		case 3:
		//parse text lines from the TG, populate page navigation structure
			paiHmiDefinePageNavigation(p);

			//define current top left menu
			menuTopLFSetCurrent(p);

			//set current tab
			menuTabSetCurrent(p, 1);

			p->keys.currentMenuLF = -1;
			p->prv.state = 4;
		 	p->prv.initDone = 1;
		break;
		case 4:

		break;
	}

}

//logic to handle external page changes (i.e. from the code or VC)
//when such page change takes place, button and tab need adjustment in order to keep it in sync with the new page
static void	menuCyclicExternPageChange(paiHmiTemplate_typ* p)
{
int btnIndex;
int tabIndex;
int found;

	if(!p){
		return;
	}

	if(p->runtime.pageChange != -1){
		return;//page change in progress, nothing to do
	}

	if(p->prv.pageSetByLFMenu == p->runtime.pageCurrent){
		return;//no external page changes
	}
	//exteren page change event! > adjust menu button and tabs!
	//in order to ajdust menu buttons and tabs, need to find a menu button index/tab index pair for the newly selected page index
	found = 0;

	for(btnIndex = 0; btnIndex < paiHMI_ENUM_MENU_ITEMS_LT; btnIndex++){

		for(tabIndex=0; tabIndex < paiHMI_ENUM_TABS_MAXIDX; tabIndex++){
			if(p->prv.menuLF[btnIndex].tabs[tabIndex].jumpPageId == p->runtime.pageCurrent){
				found = 1;
				break;
			}
		}

		if(found)
			break;
	}

	if(!found){
		//IMPORTANT CASE: we have not found a page that is associated with LF menu/tabs operation
		//don't do anything!
		//Explanation: in this case, a change page was made to a page outside of the scope of LF menu/tabs navigation
		//for example, screen saver could be activated, etc. allow this to take place!!!

		return;
	}

	p->prv.pageSetByLFMenu = p->runtime.pageCurrent;

	//adjust LF menu
	p->keys.currentMenuLF = btnIndex;
	menuCyclicKeysLF(p);

	//adjust tabs
	p->keys.tabKeysRadioDataPoint = tabIndex;
	menuCyclicTabKeys(p);
}

void paiHmiPageNavLFMenuTabsCyclic(paiHmiTemplate_typ* p, char* pVisuName, UDINT indexOfTGForHmiNavigation)
{
	if(!p)
		return;

	//On system init, parse page navigation Text Group (TG) and build the page navigation structure
	paiHmiParsePageNavigationTG(p, pVisuName, indexOfTGForHmiNavigation);

	if(!p->prv.initDone)
		return;

	menuCyclicExternPageChange(p);

	menuCyclicKeysLF(p);

	menuCyclicTabKeys(p);

}
//eof
```

#### paiHmiMsgScrolling.c
```c
/********************************************************************
 * COPYRIGHT --
 ********************************************************************
 * Package: paiHmiTemplate
 * File: paiHmiMsgScrolling.c
 * Author: goran
 * Created: July 29, 2015
 *******************************************************************/

#include <bur/plctypes.h>
#ifdef _DEFAULT_INCLUDES
	#include <AsDefault.h>
#endif

/*
###############################################################################
Message scrolling support
###############################################################################
*/
static DINT paiHmiMsgScrollingGetNext(paiHmiMsgScrolling_typ* p, UDINT startIndex)
{
	int ii, jj;
	BOOL* pAlarm;

	if(!p)
		return -1;

	pAlarm = (BOOL*)p->iAdrAlarmArray;

	for(ii=0, jj=startIndex; ii < p->iAlarmArrayLen; ii++){
		if( *(pAlarm + jj) ){
			return jj;
		}
		if(++jj>=p->iAlarmArrayLen){
			jj=0;
		}
	}
	return -1;
}

void paiHmiMsgScrollingInit(paiHmiMsgScrolling_typ* p, UDINT pAlarmArray, UDINT alarmArrayLen, UDINT msgTimeXms)
{
	if(!p)
		return;

	p->iAdrAlarmArray = (UDINT) pAlarmArray;
	p->iAlarmArrayLen = alarmArrayLen;
	p->iMsgTimeXms = msgTimeXms;
	p->state = 0; //msg not active
	p->oMsgID = 0;
	p->oMsgVisible = 1; //msg not visibile
}

void paiHmiMsgScrollingCyclic(paiHmiMsgScrolling_typ* p)
{
	int ii;
	BOOL* pAlarm;

	if(!p)
		return;

	pAlarm = (BOOL*)p->iAdrAlarmArray;

	//operate timer
	bgTimerCyclic(&p->tmr1) ;

	if(!p->iEnable){
		p->oMsgID = 0;
		p->state = 0;
		p->oMsgVisible = 1;
		return;
	}

	//if msg not active, keep searching until it becomes active
	if(!p->state){
		if( (ii = paiHmiMsgScrollingGetNext(p, 0)) < 0){
			return;
		}
		p->oMsgID = ii;
		p->state = 1;
		p->oMsgVisible = 0;
		bgTimerStart(&p->tmr1, p->iMsgTimeXms);
		return;
	}

	//timer not expired and the same alarm still active > wait
	if( !bgTimerIsTimeOut(&p->tmr1) && *(pAlarm + p->oMsgID) ){
		return;
	}

	//timer expired or msg not active any longer > find next msg to show
	if( (ii = paiHmiMsgScrollingGetNext(p, p->oMsgID + 1)) < 0){
		p->oMsgID = 0;
		p->state = 0;
		p->oMsgVisible = 1;
		return;
	}

	//show next msg
	p->oMsgID = ii;
	p->state = 1;
	p->oMsgVisible = 0;
	bgTimerStart(&p->tmr1, p->iMsgTimeXms);
}
//EOF
```

#### paiHmiPageChange.c
```c
/********************************************************************
 * COPYRIGHT -- pai
 ********************************************************************
 * Program: hmilogic
 * File: hmiAlert.c
 * Author: goran
 * Created: September 05, 2013
 *******************************************************************/

#include <bur/plctypes.h>
#ifdef _DEFAULT_INCLUDES
	#include <AsDefault.h>
#endif

void paiHmiPageChangeInit(paiHmiTemplate_typ* p)
{

}

void paiHmiPageChangeCyclic(paiHmiTemplate_typ* pHmi)
{
	if(!pHmi)
		return;

	//change screen is in progress; wait
	if( (UINT)pHmi->runtime.pageChange != 0xFFFF)
		return;

	//generate page init/exit events
	pHmi->prv.pageInit = 0;
	pHmi->prv.pageExit = 0;

	if(pHmi->runtime.pageCurrent != pHmi->prv.pagePrev){
		pHmi->prv.pageInit = 1;
		pHmi->prv.pagePrev = pHmi->runtime.pageCurrent;

	}

}
//eof
```

#### paiHmiSystemNetworking.c
```c
/********************************************************************
 * COPYRIGHT -- pai
 ********************************************************************
 * Program: hmilogic
 * File: hmiAlert.c
 * Author: goran
 * Created: September 05, 2013
 *******************************************************************/

#include <bur/plctypes.h>
#ifdef _DEFAULT_INCLUDES
	#include <AsDefault.h>
#endif

static void paiConvertIpAddrStrToDigits(char* ipAddr, USINT* pDigits);

/*
retrieve ip cfg from the device (current values)
*/
static int paiGetDeviceIpCfgData(paiHmiSystemNetworking_typ* p)
{
paiARNetworkAddress_typ* pNWCfg;
char errorText[32];
int ret_value = 0;

	if(!p)
		return -1;

	if(!p->iPtrNWConfig){
		p->oError = 1;
		brsstrcpy((UDINT)p->oErrorText, (UDINT)"iPtrNWConfig=???");
		return -1;
	}

	pNWCfg = p->iPtrNWConfig;
	brsstrcpy((UDINT)p->oCurrentNWSettings.ethDevice, (UDINT)pNWCfg->ethDevice);

	p->mGetIpAddr.enable = 1;
	p->mGetIpAddr.pDevice = (UDINT)p->oCurrentNWSettings.ethDevice;
	p->mGetIpAddr.pIPAddr = (UDINT)p->oCurrentNWSettings.ipAddr;
	p->mGetIpAddr.Len = sizeof(p->oCurrentNWSettings.ipAddr);
	CfgGetIPAddr(&p->mGetIpAddr);

	p->mGetSubnetMask.enable = 1;
	p->mGetSubnetMask.pDevice = (UDINT)p->oCurrentNWSettings.ethDevice;
	p->mGetSubnetMask.pSubnetMask = (UDINT)p->oCurrentNWSettings.netMask;
	p->mGetSubnetMask.Len = sizeof(p->oCurrentNWSettings.netMask);
	CfgGetSubnetMask(&p->mGetSubnetMask);

	p->mGetBroadcastAddr.enable = 1;
	p->mGetBroadcastAddr.pDevice = (UDINT)p->oCurrentNWSettings.ethDevice;
	p->mGetBroadcastAddr.pBroadcastAddr = (UDINT)p->oCurrentNWSettings.broadcast;
	p->mGetBroadcastAddr.Len = sizeof(p->oCurrentNWSettings.broadcast);
	CfgGetBroadcastAddr(&p->mGetBroadcastAddr);

	p->mGetDefaultGateway.enable = 1;
	p->mGetDefaultGateway.pDevice = (UDINT)p->oCurrentNWSettings.ethDevice;
	p->mGetDefaultGateway.pGateway = (UDINT)p->oCurrentNWSettings.gateway;
	p->mGetDefaultGateway.Len = sizeof(p->oCurrentNWSettings.gateway);
	CfgGetDefaultGateway(&p->mGetDefaultGateway);

	p->mGetHostName.enable = 1;
	p->mGetHostName.pHostName = (UDINT)p->oCurrentNWSettings.hostname;
	p->mGetHostName.Len = sizeof(p->oCurrentNWSettings.hostname);
	CfgGetHostName(&p->mGetHostName);

	if( (p->mGetIpAddr.status == ERR_FUB_BUSY) ||
		(p->mGetSubnetMask.status == ERR_FUB_BUSY) ||
		(p->mGetBroadcastAddr.status == ERR_FUB_BUSY) ||
		(p->mGetHostName.status == ERR_FUB_BUSY) ||
		(p->mGetDefaultGateway.status == ERR_FUB_BUSY)
	){
		return 1; //wait
	}

	if( (p->mGetIpAddr.status == ERR_OK) &&
		(p->mGetSubnetMask.status == ERR_OK) &&
		(p->mGetBroadcastAddr.status == ERR_OK) &&
		(p->mGetHostName.status == ERR_OK) &&
		(p->mGetDefaultGateway.status == ERR_OK)
	){
		p->oError = 0;
		p->oErrorText[0] = 0;
		ret_value = 0; //done; no errors
		goto exit_label;
	}

	p->oError = 2;
	p->oErrorText[0] = 0;
	if(p->mGetIpAddr.status != ERR_OK){
		brsitoa((UDINT)p->mGetIpAddr.status , (UDINT)errorText);
		brsstrcat((UDINT)p->oErrorText, (UDINT)"ipaddr=");
		brsstrcat((UDINT)p->oErrorText, (UDINT)errorText);
		brsstrcat((UDINT)p->oErrorText, (UDINT)",");
	}
	if(p->mGetSubnetMask.status != ERR_OK){
		brsitoa((UDINT)p->mGetSubnetMask.status , (UDINT)errorText);
		brsstrcat((UDINT)p->oErrorText, (UDINT)"mask=");
		brsstrcat((UDINT)p->oErrorText, (UDINT)errorText);
		brsstrcat((UDINT)p->oErrorText, (UDINT)",");
	}
	if(p->mGetBroadcastAddr.status != ERR_OK){
		brsitoa((UDINT)p->mGetBroadcastAddr.status , (UDINT)errorText);
		brsstrcat((UDINT)p->oErrorText, (UDINT)"bcast=");
		brsstrcat((UDINT)p->oErrorText, (UDINT)errorText);
		brsstrcat((UDINT)p->oErrorText, (UDINT)",");
		brsstrcat((UDINT)p->oCurrentNWSettings.broadcast, (UDINT)"=");
		brsstrcat((UDINT)p->oCurrentNWSettings.broadcast, (UDINT)errorText);
	}
	if(p->mGetDefaultGateway.status != ERR_OK){
		brsitoa((UDINT)p->mGetDefaultGateway.status , (UDINT)errorText);
		brsstrcat((UDINT)p->oErrorText, (UDINT)"gateway=");
		brsstrcat((UDINT)p->oErrorText, (UDINT)errorText);
		brsstrcat((UDINT)p->oErrorText, (UDINT)",");
		brsstrcat((UDINT)p->oCurrentNWSettings.gateway, (UDINT)"=");
		brsstrcat((UDINT)p->oCurrentNWSettings.gateway, (UDINT)errorText);
	}
	if(p->mGetHostName.status != ERR_OK){
		brsitoa((UDINT)p->mGetHostName.status , (UDINT)errorText);
		brsstrcat((UDINT)p->oErrorText, (UDINT)"host=");
		brsstrcat((UDINT)p->oErrorText, (UDINT)errorText);
		brsstrcat((UDINT)p->oErrorText, (UDINT)",");
	}

	ret_value = -1; //done; with errors

exit_label:

	//turn off fbk-s
	p->mGetIpAddr.enable = 0;
	CfgGetIPAddr(&p->mGetIpAddr);

	p->mGetSubnetMask.enable = 0;
	CfgGetSubnetMask(&p->mGetSubnetMask);

	p->mGetBroadcastAddr.enable = 0;
	CfgGetBroadcastAddr(&p->mGetBroadcastAddr);

	p->mGetDefaultGateway.enable = 0;
	CfgGetDefaultGateway(&p->mGetDefaultGateway);

	p->mGetHostName.enable = 0;
	CfgGetHostName(&p->mGetHostName);

	//generate numerical version for all network addresses (for HMI editing)
	paiConvertIpAddrStrToDigits(p->oCurrentNWSettings.ipAddr, p->oNumericalNWSettings.ipAddr);
	paiConvertIpAddrStrToDigits(p->oCurrentNWSettings.broadcast, p->oNumericalNWSettings.broadcast);
	paiConvertIpAddrStrToDigits(p->oCurrentNWSettings.gateway, p->oNumericalNWSettings.gateway);
	paiConvertIpAddrStrToDigits(p->oCurrentNWSettings.netMask, p->oNumericalNWSettings.netMask);

	return ret_value;
}
#if 0

/*
set device ip cfg data
*/
static int paiCfgSetDeviceIpCfgData(paiHmiSystemNetworking_typ* p)
{
	return 0;
  if(cfg->setIpAddr.status == 0xFFFF)   {               //  WBR:  set in previous state if cfgIP != devIP
  // if( cfg->cfgIP->addr[0] ){
    cfg->setIpAddr.enable = 1;
    cfg->setIpAddr.pDevice = (UDINT)cfg->ethDevice;
    cfg->setIpAddr.pIPAddr = (UDINT)&cfg->cfgIP->addr[0];
    cfg->setIpAddr.Option = 1;
    CfgSetIPAddr(&cfg->setIpAddr);

    if(cfg->setIpAddr.status == 0xFFFF)   return  1;
  }

  if(cfg->setBroadcastAddr.status == 0xFFFF)   {
  // if( cfg->cfgIP->broadcast[0] ){
    cfg->setBroadcastAddr.enable = 1;
    cfg->setBroadcastAddr.pDevice = (UDINT)cfg->ethDevice;
    cfg->setBroadcastAddr.pBroadcastAddr = (UDINT)&cfg->cfgIP->broadcast[0];       // WBR:  disable for CP1382 until CfgSetBroadcastAddr is fixed in the AR > 4.0
    cfg->setBroadcastAddr.Option = 1;
    CfgSetBroadcastAddr(&cfg->setBroadcastAddr);

    if(cfg->setBroadcastAddr.status == 0xFFFF)   return  1;
  }

  if(cfg->setDefaultGateway.status == 0xFFFF)   {
  // if( cfg->cfgIP->gateway[0] ){
    cfg->setDefaultGateway.enable = 1;
    cfg->setDefaultGateway.pDevice = (UDINT)cfg->ethDevice;
    cfg->setDefaultGateway.pGateway= (UDINT)&cfg->cfgIP->gateway[0];
    cfg->setDefaultGateway.Option = 1;
    CfgSetDefaultGateway(&cfg->setDefaultGateway);

    if(cfg->setDefaultGateway.status == 0xFFFF)   return  1;
  }

  if(cfg->setSubnetMask.status == 0xFFFF)   {
  // if( cfg->cfgIP->subnet[0] ){
    cfg->setSubnetMask.enable = 1;
    cfg->setSubnetMask.pDevice = (UDINT)cfg->ethDevice;
    cfg->setSubnetMask.pSubnetMask = (UDINT)&cfg->cfgIP->subnet[0];
    cfg->setSubnetMask.Option = 1;
    CfgSetSubnetMask(&cfg->setSubnetMask);

    if(cfg->setSubnetMask.status == 0xFFFF)   return  1;
  }

  if  (   (cfg->setIpAddr.status == 65535) ||
      (cfg->setSubnetMask.status == 65535) ||
      (cfg->setBroadcastAddr.status == 65535) ||
      (cfg->setDefaultGateway.status == 65535)
    ){
    return 1;
  }

  if  (   !cfg->getIpAddr.status &&
      !cfg->setSubnetMask.status &&
      !cfg->setBroadcastAddr.status &&
      !cfg->setDefaultGateway.status
    ){

    // DBG("setDeviceIpCfg: IpAddr='%s'\r\n", cfg->cfgIP->addr);
    // DBG("setDeviceIpCfg: SubnetMask='%s'\r\n", cfg->cfgIP->subnet);
    // DBG("setDeviceIpCfg: BroadcastAddr='%s'\r\n", cfg->cfgIP->broadcast);
    // DBG("setDeviceIpCfg: DefaultGateway='%s'\r\n", cfg->cfgIP->gateway);

    return 0;
  }

  // DBG("setDeviceIpCfg: ERROR\r\n");
  // DBG("setDeviceIpCfg: IpAddr='%s'  st=%d\r\n", cfg->cfgIP->addr, cfg->getIpAddr.status);
  // DBG("setDeviceIpCfg: SubnetMask='%s'  st=%d\r\n", cfg->cfgIP->subnet, cfg->setSubnetMask.status);
  // DBG("setDeviceIpCfg: BroadcastAddr='%s'  st=%d\r\n", cfg->cfgIP->broadcast, cfg->setBroadcastAddr.status);
  // DBG("setDeviceIpCfg: DefaultGateway='%s'  st=%d\r\n", cfg->cfgIP->gateway, cfg->setDefaultGateway.status);

  return -1;
}
#endif
#if 0

static int paiCfgCompareDeviceAndFileCfgData(paiHmiSystemNetworking_typ* p)
{
	return 0;
 int update = 0;     //! \todo   assign update with flags to indicate settings that need to change

  if(cfg->cfgIP->addr[0] && ( strcmp(&cfg->cfgIP->addr[0], &cfg->devIP.addr[0]) ))  {
    // DBGINF("Cfg update needed: cfgIP->addr='%s' devIP.addr='%s'\r\n", &cfg->cfgIP->addr[0], &cfg->devIP.addr[0]);
    cfg->setIpAddr.status=  0xFFFF;
    update = 1;
  }

  if(cfg->cfgIP->subnet[0] && ( strcmp(&cfg->cfgIP->subnet[0], &cfg->devIP.subnet[0]) ))  {
    // DBGINF("Cfg update needed: cfgIP->subnet='%s' devIP.subnet='%s'\r\n", &cfg->cfgIP->subnet[0], &cfg->devIP.subnet[0]);
    cfg->setSubnetMask.status=  0xFFFF;
    update = 1;
  }

#ifdef  AS_CFG
  if(!strcmp("PP420_1043_K27", AS_CFG))   {
    if(cfg->cfgIP->broadcast[0] && ( strcmp(&cfg->cfgIP->broadcast[0], &cfg->devIP.broadcast[0]) ))   {
      // DBGINF("Cfg update needed: cfgIP->broadcast='%s' devIP.broadcast='%s'\r\n", &cfg->cfgIP->broadcast[0], &cfg->devIP.broadcast[0]);
      cfg->setBroadcastAddr.status=  0xFFFF;
      update = 1;
    }
  }
#endif

  if(cfg->cfgIP->gateway[0] && ( strcmp(&cfg->cfgIP->gateway[0], &cfg->devIP.gateway[0]) ))   {
    // DBGINF("Cfg update needed: cfgIP->gateway='%s' devIP.gateway='%s'\r\n", &cfg->cfgIP->gateway[0], &cfg->devIP.gateway[0]);
    cfg->setDefaultGateway.status=  0xFFFF;
    update = 1;
  }

  return update;
}
#endif

static void paiConvertIpAddrStrToDigits(char* ipAddr, USINT* pDigits)
{
//"127.0.0.1" --> digit[0]=127; digit[1]=0; digit[2]=0; digit[3]=1
char txtIpAddr[32];
char txtDigit[4][8];
int ii;
int jj;
char* pBeg;

	brsstrcpy((UDINT)txtIpAddr, (UDINT)ipAddr);
	txtDigit[0][0] = 0;
	txtDigit[1][0] = 0;
	txtDigit[2][0] = 0;
	txtDigit[3][0] = 0;

	pBeg = txtIpAddr;
	for(ii=0, jj=0; jj < 32; jj++){
		if(txtIpAddr[jj] == '.'){
			txtIpAddr[jj] = 0;
			brsstrcpy((UDINT)txtDigit[ii++], (UDINT)pBeg);
			pBeg = &txtIpAddr[jj+1];
			if(ii >= 3){
				brsstrcpy((UDINT)txtDigit[ii], (UDINT)pBeg);
				break;
			}
		}
	}

	for(ii=0; ii < 4; ii++){
		*pDigits = (USINT)brsatoi((UDINT)txtDigit[ii]);
		pDigits++;
	}
}
#if 0
static void paiConvertIpDigitsToIpAddrStr(char* ipAddr, USINT* pDigits)
{
char txtDigit[8];
char txtIpAddr[32];

	if(!ipAddr || !pDigits)
		return;

	txtIpAddr[0] = 0;

	brsitoa((UDINT)pDigits[0], (UDINT)txtDigit);
	brsstrcat((UDINT)txtIpAddr, (UDINT)txtDigit);
	brsstrcat((UDINT)txtIpAddr, (UDINT)".");

	brsitoa((UDINT)pDigits[1], (UDINT)txtDigit);
	brsstrcat((UDINT)txtIpAddr, (UDINT)txtDigit);
	brsstrcat((UDINT)txtIpAddr, (UDINT)".");

	brsitoa((UDINT)pDigits[2], (UDINT)txtDigit);
	brsstrcat((UDINT)txtIpAddr, (UDINT)txtDigit);
	brsstrcat((UDINT)txtIpAddr, (UDINT)".");

	brsitoa((UDINT)pDigits[3], (UDINT)txtDigit);
	brsstrcat((UDINT)txtIpAddr, (UDINT)txtDigit);

}
#endif

void paiHmiSystemNetworkingInit(paiHmiSystemNetworking_typ* p)
{
	p->oError = 0; //no errors
	p->oErrorText[0] = 0; //no errors
	p->oState = 1; //get current settings
}

void paiHmiSystemNetworkingCyclic(paiHmiSystemNetworking_typ* p)
{
	switch(p->oState){
		case 1:
			if( paiGetDeviceIpCfgData(p) == 1 )
				return; //wait

			p->oState = 0;//done
		break;
		default:
			p->oState = 0;
		break;
	}
}
//eof
```

#### paiHmiTableViewPersons.c
```c
/********************************************************************
 * COPYRIGHT -- pai
 ********************************************************************
 * Program: hmilogic
 * File: hmiTableViewPersons.c
 * Author: goran
 * Created: November 24, 2013
 ********************************************************************
 * Implementation of program hmiTableViewPersons
 ********************************************************************/

#include <bur/plctypes.h>

#ifdef _DEFAULT_INCLUDES
	#include <AsDefault.h>
#endif

/**
Bit manipulaiton utility functions.
 */
//#include <../../bglib/bgBitUtilities.h>

/**
String manipulaiton utility functions.
 */
#include <../../bglib/bgsprintf.h>
//#include <../../bglib/bgstring.h>

//#include <../../RecFIFO/fifotest/fifoif.h>

/*
###############################################################################
Table View support functions
###############################################################################
*/

/*
Display table background grid (i.e. each odd row in one color, each even row in
a different color
*/
void tableViewShowGrid(hmiTablePersons_typ* p)
{
	int ii;

	for(ii=0; ii<=p->viewIndexMax; ii++){
		//select a different collor scheme for each row of the table
		if(ii%2){
			p->itemsInView[ii].ctrl.bgdColorIndex = 1;
		}else{
			p->itemsInView[ii].ctrl.bgdColorIndex = 0;
		}
	}
}

/*
Init table based person viewer
*/
void tableViewPersonsInit(hmiTablePersons_typ* p, hmiTableItemDataPerson_typ* pItemsAll, UDINT itemCount, UDINT viewIndexMax, char* pDBTableName, int jsonSQLQueryid)
{
	int ii;

	if(!p || !pItemsAll || !itemCount || !viewIndexMax)
		return;

	p->pItemsAll = (UDINT)pItemsAll;

	p->viewIndexMax = viewIndexMax;
	if(p->viewIndexMax > hmiTablePersonMAXVIEWINDEX){
		p->viewIndexMax = hmiTablePersonMAXVIEWINDEX;
	}
	p->viewIndex = 0;

	tableViewShowGrid(p);

	//reset selection/activate indexes and datapoints wired to hotspots
	p->selectedItem = -1;
	p->selectedViewItem = -1;
	p->selectViewItemDataPoint = -1;
	p->activateViewItemDataPoint = -1;
	if(pDBTableName)
		brsstrcpy((UDINT)p->activeDBTableName, (UDINT)pDBTableName);
	p->activeSQLid = jsonSQLQueryid;

	p->itemCountUnfiltered = 0;
	p->itemCount = 0;
	for(ii=0; ii<itemCount;ii++){
		if(pItemsAll[ii].usedEntry){
			p->itemCountUnfiltered++;
			p->itemCount++;
		}
	}
}

/*
Hide (don't show) table row data at a selected row. Result is an empty line.
*/
static void personTableHideItemAtIndex(hmiTablePersons_typ* p, int viewIndex)
{
	if(!p || viewIndex > p->viewIndexMax)
		return;
	p->itemsInView[viewIndex].ctrl.visibilityControl = 1;
}

/*
Show (don't hide) table row data at a selected row. Result is an line that contais all columns (i.e. text fields).
*/
static void personTableShowItemAtIndex(hmiTablePersons_typ* p, int viewIndex)
{
	if(!p || viewIndex > p->viewIndexMax)
		return;

	//convert numerics into txt
	bgsprintf(p->itemsInView[viewIndex].data.employeeIdTxt, "%d", p->itemsInView[viewIndex].data.employeeId);
	bgsprintf(p->itemsInView[viewIndex].data.indexTxt, "%d", p->itemsInView[viewIndex].data.index);
	bgsprintf(p->itemsInView[viewIndex].data.shiftTxt, "%d", p->itemsInView[viewIndex].data.shift);

	//make item visible
	p->itemsInView[viewIndex].ctrl.visibilityControl = 0;
}

/*
Display table view.
*/
void tableViewShow(hmiTablePersons_typ* p)
{
	int ii, jj;
	hmiTableItemDataPerson_typ* pItemsAll;

	if(!p || !p->pItemsAll)
		return;

	pItemsAll = (hmiTableItemDataPerson_typ*)p->pItemsAll;

	for(ii=0, jj = p->viewIndex; ii<=p->viewIndexMax; jj++){
		if(pItemsAll[jj].index < 0)
			continue;

		if(jj<p->itemCountUnfiltered){
			brsmemcpy((UDINT)&p->itemsInView[ii].data, (UDINT)&pItemsAll[jj], sizeof(hmiTableItemDataPerson_typ) );
			personTableShowItemAtIndex(p, ii);
		}else{
			personTableHideItemAtIndex(p, ii);
		}
		ii++;
	}
}

/*
Selection (i.e. row highlighting) of the table row.
*/
static void tableViewItemSelection(hmiTablePersons_typ* p)
{
	if(!p)
		return;

	//table item selection logic
	//selectViewItemDataPoint is connected to a hotstop above the table line. Each line sets a different
	//number that corepsonds to the visible (table) line number.
	if( (p->selectViewItemDataPoint >= 0) && (p->selectViewItemDataPoint <= p->viewIndexMax)){
		//check if a table line is already selected
		if(p->selectedViewItem < 0){
			//no item selected > select it now
			p->selectedViewItem = p->selectViewItemDataPoint; //save selected line for lated
			p->bgdColorIndexOldSelection = p->itemsInView[p->selectedViewItem].ctrl.bgdColorIndex;//save current color index for the line to be able to restore it
			p->itemsInView[p->selectedViewItem].ctrl.bgdColorIndex = 2;//select 3-rd color from the map
			//save current selection
			p->selectedViewItem = p->selectViewItemDataPoint;
		}else
			if(p->selectedViewItem == p->selectViewItemDataPoint){
			//same item is already selected > deselect it now (toggle selection)
			//restore background color for the line
			p->itemsInView[p->selectedViewItem].ctrl.bgdColorIndex = p->bgdColorIndexOldSelection;
			//reset selection status
			p->selectedViewItem = -1;
		}else{
			//deactivate old selection, activate new selection
			p->itemsInView[p->selectedViewItem].ctrl.bgdColorIndex = p->bgdColorIndexOldSelection;
			p->bgdColorIndexOldSelection = p->itemsInView[p->selectViewItemDataPoint].ctrl.bgdColorIndex;
			p->itemsInView[p->selectViewItemDataPoint].ctrl.bgdColorIndex = 2;
			//save current selection
			p->selectedViewItem = p->selectViewItemDataPoint;
		}

		//calculate a line from the entire table that is currently selected
		p->selectedItem = -1;
		if(p->selectedViewItem >= 0)
			p->selectedItem = p->selectedViewItem + p->viewIndex;

		//reset datapoint connected to hotspots
		p->selectViewItemDataPoint = -1;
	}
}

/*
Logic to set / reset an "active" property (i.e. column) of a persons table
*/
static void tableViewItemActive(hmiTablePersons_typ* p)
{
	UDINT rawIndex;
	hmiTableItemDataPerson_typ* pItemsAll;

	if(!p || !p->pItemsAll)
		return;

	return;//TODO: disable section below until a full support is available; that way, changing activ/inactive button on the
	//worker / inspector screen would not be working at all (instead of giving a false impression that the tnings are working)

	pItemsAll = (hmiTableItemDataPerson_typ*)p->pItemsAll;
	//table item active/inactive logic
	//activateViewItemDataPoint is connected to a hotstop above the active field within a table line. Each line sets a different
	//number that corepsonds to the visible (table) line number.
	if( (p->activateViewItemDataPoint >= 0) && (p->activateViewItemDataPoint <= p->viewIndexMax)){
		//check if a table line is already active
		if(p->itemsInView[p->activateViewItemDataPoint].data.active){
			p->itemsInView[p->activateViewItemDataPoint].data.active = 0;
			rawIndex = p->itemsInView[p->activateViewItemDataPoint].data.indexRaw;
			pItemsAll[rawIndex].active = 0;
			//execute DB update

		}else{
			p->itemsInView[p->activateViewItemDataPoint].data.active = 1;
			rawIndex = p->itemsInView[p->activateViewItemDataPoint].data.indexRaw;
			pItemsAll[rawIndex].active = 1;
			//execute DB update

		}
		p->activateViewItemDataPoint = -1;
	}
}

static void tableViewRefresh(hmiTablePersons_typ* p)
{
	p->selectedViewItem = -1;//invalidate view selection for a proper redraw of the selected item
	tableViewShowGrid(p); //redraw table layout
	tableViewShow(p); //redraw table data
}

static void tableViewScroll(hmiTablePersons_typ* p)
{
	if(!p || !p->itemCount)
		return;

	//if no item is selected, and any scroll key pressed, just select a top item on the list
	if( (p->selectedItem < 0) &&
		(p->btnScrollLineUp || p->btnScrollPageUp || p->btnScrollLineDw || p->btnScrollPageDw)){
		p->btnScrollLineUp = 0; p->btnScrollPageUp = 0;
		p->btnScrollLineDw = 0; p->btnScrollPageDw = 0;
		//item is NOT selected > select the top item
		p->selectViewItemDataPoint = 0;
		tableViewItemSelection(p);
		return;
	}

	//table scroll logic
	if(p->btnScrollLineUp){
		p->btnScrollLineUp = 0;

		if(!p->selectedItem){
			return;//top item is already selected > nothing to do
		}

		if(!p->selectedViewItem){
			//selected view item is at the TOP
			//is the view index > 0 (which means that scroll window has a chance to to move up)
			if(p->viewIndex){
				//view index is not all the way up > scroll it up
				p->viewIndex--;
				tableViewRefresh(p);//display the entire table
			}
			p->selectViewItemDataPoint = 0;//select the top line in the view
		}else{
			//selected view item is not the TOP > need to scroll up selection within the visible view
			p->selectViewItemDataPoint = p->selectedViewItem -  1;
		}
		//update selection
		tableViewItemSelection(p);
		return;
	}

	if(p->btnScrollLineDw){
		p->btnScrollLineDw = 0;

		//item is already selected > scroll line dw
		if(p->selectedItem == (p->itemCount - 1)){
			//last item is already selected
			return;
		}

		if(p->selectedViewItem >= p->viewIndexMax){
			//selected view item is the LAST item in the view
			if(p->viewIndex < (p->itemCount - (p->viewIndexMax + 1) ) ){
				//view index can be further moved  > scroll
				p->viewIndex++;
				tableViewRefresh(p);
			}
			p->selectViewItemDataPoint = p->viewIndexMax;//select last item in the table view
		}else{
			//selected view item is not the BOTTOM > scroll
			p->selectViewItemDataPoint = p->selectedViewItem +  1;
		}
		tableViewItemSelection(p);
		return;
	}

	if(p->btnScrollPageUp){
		p->btnScrollPageUp = 0;

		//is view window at the top?
		if(p->viewIndex){
			//no > scroll up by the page size
			p->viewIndex -= p->viewIndexMax+1;
			//viewIndex cann't be < 0!
			if(p->viewIndex < 0){
				p->viewIndex = 0;
				p->selectViewItemDataPoint = 0;
			}else{
				p->selectViewItemDataPoint = p->selectedViewItem;
			}
			tableViewRefresh(p);//display the entire table
		}else{
			//view window is alreday all the way up > select the top line on the view
			if(p->selectedViewItem)
				p->selectViewItemDataPoint = 0;
		}
		//redraw selection
		tableViewItemSelection(p);
		return;
	}

	if(p->btnScrollPageDw){
		p->btnScrollPageDw = 0;

		//is the selection at the bottom?
		if((p->itemCount -1) <= p->selectedItem){
			//view window is alreday all the way dw > select the bottom line on the view
			return;
		}

		//no > scroll dw by the page size
		if( ((p->itemCount) / (p->viewIndexMax+1)) > ((p->selectedItem + 1) / (p->viewIndexMax+1))){
			p->viewIndex += p->viewIndexMax+1;
			if(p->viewIndex > (p->itemCount - 1 )){
				p->viewIndex = (p->itemCount - 1);
			}
			//p->selectViewItemDataPoint = p->selectedViewItem;
			p->selectViewItemDataPoint = 0;
			tableViewRefresh(p);
		}

		//redraw selection
		tableViewItemSelection(p);
		return;
	}

}

/*
Persons table view filter
shiftFilter - 0-show all (both shifts);1-shift1;2-shift2
activeFilger - 0-show all (active and not active); 1-show active only
*/
void tableFilterPersonsSet(hmiTablePersons_typ* p, int shiftFilter, int activeFilter, int assignedFilter)
{
	if(!p)
		return;

	p->shiftFilter = 0;//default: no filtering on shift
	if( (shiftFilter >= 0) && (shiftFilter <= 2)){
		p->shiftFilter = shiftFilter;
	}

	p->activeFilter = 0;//default: no filtering on active
	if( (activeFilter >= 0) && (activeFilter <= 1)){
		p->activeFilter = activeFilter;
	}

	p->assignedFilter = 0;//default: no filtering on person assigned to a station
	if( (assignedFilter >= 0) && (assignedFilter <= 1)){
		p->assignedFilter = assignedFilter;
	}

}

void tableFilterExecute(hmiTablePersons_typ* p)
{
	if(!p)
		return;

	p->executeFilter = 1;//execute filter request; cleared upon filter execution
}

int tableFilterPersonsActive(hmiTableItemDataPerson_typ* pItem, int activeFilter)
{
	if(activeFilter == 1){
		//pass only active items
		if(pItem->active == 1){
			return 1;
		}
		return 0;
	}

	return 1;//pass all items
}

int tableFilterPersonsShift(hmiTableItemDataPerson_typ* pItem, int shiftFilter)
{
	switch(shiftFilter){
		case 1://pass shift 1 only items
			if(pItem->shift == 1){
				return 1;
			}
			return 0;
		break;
		case 2://pass shift 2 only items
			if(pItem->shift == 2){
				return 1;
			}
			return 0;
		break;
		default:
		break;
	}
	return 1;//pass all items
}

static int tableFilterIsUpdate(hmiTablePersons_typ* p, int* filterType)
{
	int filterLocal = 0;
	int filterDB = 0;

	if(!p){
		if(filterType)
			*filterType = 0;
		return 0;
	}

	//filter setting changed?
	if( !p->executeFilter &&
		(p->shiftFilter == p->shiftFilterOld) &&
		(p->activeFilter == p->activeFilterOld) &&
		(p->assignedFilter == p->assignedFilterOld) &&
		(p->azFilterFirstName == p->azFilterFirstNameOld) &&
		(p->azFilterLastName == p->azFilterLastNameOld)
	){
		//no changes for filters that required DB request
	}else{
		filterDB = 1;
	}

	if( (p->assignedFilter == p->assignedFilterOld) ){
		//no changes for filters that are performed localy
	}else{
		filterLocal = 1;
	}

	p->executeFilter = 0;
	p->shiftFilterOld = p->shiftFilter;
	p->activeFilterOld = p->activeFilter;
	p->assignedFilterOld = p->assignedFilter;
	p->azFilterLastNameOld = p->azFilterLastName;
	p->azFilterFirstNameOld = p->azFilterFirstName;

	*filterType = filterDB + (2 * filterLocal);//bit0-filterDB, bit1-filterLocal

	return 1;
}

/*
SELECT id,lastname,firstname,employeeid,active,shift FROM workers  ORDER BY lastname,firstname

SELECT id,lastname,firstname,employeeid,active,shift FROM workers  WHERE  active = 1  AND  shift = 1  ORDER BY lastname  ,firstname
SELECT id,lastname,firstname,employeeid,active,shift FROM workers  WHERE  active = 1  ORDER BY lastname  ,firstname
SELECT id,lastname,firstname,employeeid,active,shift FROM workers  WHERE  active = 0  ORDER BY lastname  ,firstname
SELECT id,lastname,firstname,employeeid,active,shift FROM workers  WHERE  shift =  2 ORDER BY lastname  ,firstname
SELECT id,lastname,firstname,employeeid,active,shift FROM workers  WHERE  active = 0  AND  shift =  2 ORDER BY lastname  ,firstname

SELECT id,lastname,firstname,employeeid,active,shift FROM workers  ORDER BY lastname  ,firstname  DESC
SELECT id,lastname,firstname,employeeid,active,shift FROM workers  ORDER BY lastname  DESC  ,firstname  DESC
*/
static void tableFilterPersons(hmiTablePersons_typ* p)
{
	int filterMode;//bit0-DBfilter, bit1-localFilter

	char* pActiveFilter;
	char* pShiftFilter;
	char* pAZSortLast;
	char* pAZSortFirst;
	char textBuf[32];
	char gUdpClient_txbuf[255];

	if(!p || !p->pItemsAll)
		return;

	//check if running a filter is requested?
	if( !tableFilterIsUpdate(p, &filterMode) )
		return ;

	if(filterMode & 0x2){
		//local filter (station assigment)
		//DBG(lgr, "Apply filter: station assing");
	}

	if(!(filterMode & 0x1)){
		return;
	}

	switch(p->activeFilter){
		case 1: pActiveFilter = " active = 1 ";break;
		case 2: pActiveFilter = " active = 0 ";break;
		default:
			pActiveFilter = 0;
			break;
	}
	switch(p->shiftFilter){
		case 1: pShiftFilter = " shift = 1 ";break;
		case 2: pShiftFilter = " shift = 2 ";break;
		default:
			pShiftFilter = 0;
			break;
	}
	switch(p->azFilterLastName){
		case 1: pAZSortLast = " DESC ";break;
		default:
			pAZSortLast = 0;
			break;
	}
	switch(p->azFilterFirstName){
		case 1: pAZSortFirst = " DESC ";break;
		default:
			pAZSortFirst = 0;
			break;
	}

	brsstrcpy((UDINT)&gUdpClient_txbuf[0], (UDINT)"{\"paipvilite\": \"1.0\", \"method\": \"executesqlquery\", \"params\": {\"sqlquery\":\"SELECT id,lastname,firstname,employeeid,active,shift FROM ");
	brsstrcat((UDINT)&gUdpClient_txbuf[0], (UDINT)p->activeDBTableName);
	if(pActiveFilter || pShiftFilter){
		brsstrcat((UDINT)&gUdpClient_txbuf[0], (UDINT)" WHERE ");
		if(pActiveFilter)
			brsstrcat((UDINT)&gUdpClient_txbuf[0], (UDINT)pActiveFilter);
		if(pActiveFilter && pShiftFilter)
			brsstrcat((UDINT)&gUdpClient_txbuf[0], (UDINT)" AND ");
		if(pShiftFilter)
			brsstrcat((UDINT)&gUdpClient_txbuf[0], (UDINT)pShiftFilter);
	}

	brsstrcat((UDINT)&gUdpClient_txbuf[0], (UDINT)" ORDER BY lastname ");
	if(pAZSortLast)
		brsstrcat((UDINT)&gUdpClient_txbuf[0], (UDINT)pAZSortLast);

	brsstrcat((UDINT)&gUdpClient_txbuf[0], (UDINT)" ,firstname ");
	if(pAZSortFirst)
		brsstrcat((UDINT)&gUdpClient_txbuf[0], (UDINT)pAZSortFirst);

	brsstrcat((UDINT)&gUdpClient_txbuf[0], (UDINT)"\"}, \"id\": ");
	brsitoa(p->activeSQLid, (UDINT)textBuf);
	brsstrcat((UDINT)&gUdpClient_txbuf[0], (UDINT)textBuf);
	brsstrcat((UDINT)&gUdpClient_txbuf[0], (UDINT)"}");

	pushSQLQuery(0, (unsigned char*)gUdpClient_txbuf, brsstrlen((UDINT)gUdpClient_txbuf));

	//gUdpClient.clientIf.iSend = 1;
}

DINT tableFilterGetSelectedItemRawIndex(hmiTablePersons_typ* p, int selectedItem)
{
	DINT ii;
	hmiTableItemDataPerson_typ* pItemsAll;

	if(!p || !p->pItemsAll)
		return 0;

	pItemsAll = (hmiTableItemDataPerson_typ*)p->pItemsAll; //ptr to an array of all records
	//iterate over all records
	for(ii=0; ii<p->itemCountUnfiltered; ii++, pItemsAll++){
		if((pItemsAll->index < 0) || (pItemsAll->index != selectedItem))
			continue;
		return ii;
	}

	return -1;
}

void tablePersonsCyclic()
{
	hmiTablePersons_typ* pT = &gHmi.tableViewPersons;

	//table show view
	tableViewShow(pT);

	//table item (row) selection logic
	tableViewItemSelection(pT);

	//table item active/inactive logic
	tableViewItemActive(pT);

	//table scroll logic
	tableViewScroll(pT);

	//table filtering (i.e. shift 1 or 2, active or not active)
	tableFilterPersons(pT);
}
//EOF
```

### Program Logical/paiComponents/paiMp/paiFileDT

#### paiFileDT.var
```iecst
VAR
	ii : UDINT := 0;
END_VAR
```

#### paiFileItemDT.st
```iecst
PROGRAM _CYCLIC
	(* Insert code here *)

	//Convert DT values to string for use in VC
	FOR ii := 0 TO 9 DO
		IF(gPaiMp.data.MpFileManagerUIConnect.File.List.Items[ii].LastModified > DT#1970-01-01-00:00:00) THEN
			gPaiMp.data.paiFileItemSizeAndDT[ii].strDT := DT_TO_STRING(gPaiMp.data.MpFileManagerUIConnect.File.List.Items[ii].LastModified);
		ELSE
			gPaiMp.data.paiFileItemSizeAndDT[ii].strDT := WSTRING_TO_STRING(" ");
		END_IF
		IF(gPaiMp.data.MpFileManagerUIConnect.File.List.Items[ii].ItemType >= mpFILE_ITEM_TYPE_FILE) THEN
			gPaiMp.data.paiFileItemSizeAndDT[ii].strSize := UDINT_TO_STRING(gPaiMp.data.MpFileManagerUIConnect.File.List.Items[ii].Size);
		ELSE
			gPaiMp.data.paiFileItemSizeAndDT[ii].strSize := WSTRING_TO_STRING(" ");
		END_IF
	END_FOR;
END_PROGRAM
```

### Program Logical/paiComponents/paiMp/paiMp (ANSIC)

#### paiMp.c - Cyclic code
```c
#include <bur/plctypes.h>

#ifdef _DEFAULT_INCLUDES
	#include <AsDefault.h>
#endif

#include "../../paiFileService/paiFS/paiFile.h"

/*
###############################################################################
PAI_CONFIGURATION_SECTION
Code below allows configuration for:
mapp components used in this application
###############################################################################
*/

#warning "pai Configuration: mapp Components"

//=============================================================================
//MpCom support
//=============================================================================
static void paiMpComInit()
{

	MpComIdentType link;
	link.Internal[0] = mpCOM_MAIN_INT;

	gPaiMp.fub.MpComLoggerUI.Enable = 1;
//	gPaiMp.data.MpComIdent.Internal[0] = mpCOM_MAIN_INT;
//	gPaiMp.data.MpComIdent.Internal[1] = 0;
//	gPaiMp.fub.MpComLoggerUI.MpLink = &link;
	gPaiMp.fub.MpComLoggerUI.UIConnect = &gPaiMp.data.MpComLoggerUIConnect;

	gPaiMp.fub.MpComLoggerUI.UISetup.LoggerListSize = 8;
	gPaiMp.fub.MpComLoggerUI.UISetup.LoggerScrollWindow = 1;

	gPaiMp.fub.MpComLoggerUI.Scope = mpCOM_CONFIG_SCOPE_BRANCH;

}

static void paiMpComCyclic()
{

	MpComLoggerUI(&gPaiMp.fub.MpComLoggerUI);

}

//=============================================================================
//MpAlarm support
//=============================================================================
static void paiMpAlarmInit()
{

}

static void paiMpAlarmCyclic()
{
	MpAlarmBasicUI(&gPaiMp.fub.MpAlarmBasicUI);
}

static void paiMpRecipeInit()
{
	gPaiMp.fub.MpRecipeXml.Enable = 1;
	gPaiMp.fub.MpRecipeXml.MpLink = &gMpLinkMpRecipeXml;
	gPaiMp.fub.MpRecipeXml.DeviceName = PAI_FS_DEVICE_REC;
	gPaiMp.fub.MpRecipeXml.FileName = "recipe";

	gPaiMp.fub.MpRecipeRegPar.Enable = 1;
	gPaiMp.fub.MpRecipeRegPar.MpLink = &gMpLinkMpRecipeXml;
	gPaiMp.fub.MpRecipeRegPar.PVName = "gRecipe";

	gPaiMp.fub.MpRecipeUI.Enable = 1;
	gPaiMp.fub.MpRecipeUI.MpLink = &gMpLinkMpRecipeXml;
	gPaiMp.fub.MpRecipeUI.UISetup.RecipeListSize = 10;
	gPaiMp.fub.MpRecipeUI.UISetup.RecipeListScrollWindow = 1;
	gPaiMp.fub.MpRecipeUI.UISetup.Confirmation.RecipeCreate = 1;
	gPaiMp.fub.MpRecipeUI.UISetup.Confirmation.RecipeLoad = 1;
	gPaiMp.fub.MpRecipeUI.UISetup.Confirmation.RecipeSave = 1;

	gPaiMp.fub.MpRecipeUI.UIConnect = &gPaiMp.data.MpRecipeUIConnect;
}

static void paiMpRecipeCustom1Init()
{
	gPaiMp.fub.MpRecipeXmlCustom1.Enable = 1;
	gPaiMp.fub.MpRecipeXmlCustom1.MpLink = &gMpLinkMpRecipeXmlCustom1;
	gPaiMp.fub.MpRecipeXmlCustom1.DeviceName = PAI_FS_DEVICE_REC_LAYER;
	gPaiMp.fub.MpRecipeXmlCustom1.FileName = "recLayer";

	gPaiMp.fub.MpRecipeUICustom1.Enable = 1;
	gPaiMp.fub.MpRecipeUICustom1.MpLink = &gMpLinkMpRecipeXmlCustom1;
	gPaiMp.fub.MpRecipeUICustom1.UISetup.RecipeListSize = 10;
	gPaiMp.fub.MpRecipeUICustom1.UISetup.RecipeListScrollWindow = 1;
	gPaiMp.fub.MpRecipeUICustom1.UISetup.Confirmation.RecipeCreate = 1;
	gPaiMp.fub.MpRecipeUICustom1.UISetup.Confirmation.RecipeLoad = 1;
	gPaiMp.fub.MpRecipeUICustom1.UISetup.Confirmation.RecipeSave = 1;

	gPaiMp.fub.MpRecipeUICustom1.UIConnect = &gPaiMp.data.MpRecipeUIConnectCustom1;
}

static void paiMpRecipeCustom2Init()
{
	gPaiMp.fub.MpRecipeXmlCustom2.Enable = 1;
	gPaiMp.fub.MpRecipeXmlCustom2.MpLink = &gMpLinkMpRecipeXmlCustom2;
	gPaiMp.fub.MpRecipeXmlCustom2.DeviceName = PAI_FS_DEVICE_REC_PALLETE;
	gPaiMp.fub.MpRecipeXmlCustom2.FileName = "recPallete";

	gPaiMp.fub.MpRecipeUICustom2.Enable = 1;
	gPaiMp.fub.MpRecipeUICustom2.MpLink = &gMpLinkMpRecipeXmlCustom2;
	gPaiMp.fub.MpRecipeUICustom2.UISetup.RecipeListSize = 10;
	gPaiMp.fub.MpRecipeUICustom2.UISetup.RecipeListScrollWindow = 1;
	gPaiMp.fub.MpRecipeUICustom2.UISetup.Confirmation.RecipeCreate = 1;
	gPaiMp.fub.MpRecipeUICustom2.UISetup.Confirmation.RecipeLoad = 1;
	gPaiMp.fub.MpRecipeUICustom2.UISetup.Confirmation.RecipeSave = 1;

	gPaiMp.fub.MpRecipeUICustom2.UIConnect = &gPaiMp.data.MpRecipeUIConnectCustom2;
}

static void paiMpRecipeCyclic()
{
	MpRecipeXml(&gPaiMp.fub.MpRecipeXml);

	MpRecipeRegPar(&gPaiMp.fub.MpRecipeRegPar);

	MpRecipeUI(&gPaiMp.fub.MpRecipeUI);
}

static void paiMpRecipeCustom1Cyclic()
{
	MpRecipeXml(&gPaiMp.fub.MpRecipeXmlCustom1);

	//MpRecipeRegPar(&gPaiMp.fub.MpRecipeRegPar);

	MpRecipeUI(&gPaiMp.fub.MpRecipeUICustom1);
}

static void paiMpRecipeCustom2Cyclic()
{
	MpRecipeXml(&gPaiMp.fub.MpRecipeXmlCustom2);

	//MpRecipeRegPar(&gPaiMp.fub.MpRecipeRegPar);

	MpRecipeUI(&gPaiMp.fub.MpRecipeUICustom2);
}

//=============================================================================

static void paiMpFileManagerInit()
{
	brsstrcpy((UDINT)gPaiMp.data.MpFileManagerUIConnect.DeviceList.DeviceNames[0], (UDINT)PAI_FS_DEVICE_ROOT);
	brsstrcpy((UDINT)gPaiMp.data.MpFileManagerUIConnect.DeviceList.DeviceNames[1], (UDINT)PAI_FS_DEVICE_CFG);
	brsstrcpy((UDINT)gPaiMp.data.MpFileManagerUIConnect.DeviceList.DeviceNames[2], (UDINT)PAI_FS_DEVICE_REC);
	brsstrcpy((UDINT)gPaiMp.data.MpFileManagerUIConnect.DeviceList.DeviceNames[3], (UDINT)"USB1");
	brsstrcpy((UDINT)gPaiMp.data.MpFileManagerUIConnect.DeviceList.DeviceNames[4], (UDINT)"USB2");

	gPaiMp.fub.MpFileManagerUI.Enable = 1;
	gPaiMp.fub.MpFileManagerUI.MpLink = &gMpLinkMpFileManagerUI;
	gPaiMp.fub.MpFileManagerUI.UIConnect = &gPaiMp.data.MpFileManagerUIConnect;
	gPaiMp.fub.MpFileManagerUI.UISetup.FileListScrollWindow = 1;
	gPaiMp.fub.MpFileManagerUI.UISetup.FileListSize = 8;

}

static void paiMpFileManagerCyclic()
{
	MpFileManagerUI(&gPaiMp.fub.MpFileManagerUI);
}
//=============================================================================

void _INIT paiMpInit(void)
{
	paiMpComInit();

	paiMpFileManagerInit();

	paiMpRecipeInit();
	paiMpRecipeCustom1Init();
	paiMpRecipeCustom2Init();

	paiMpAlarmInit();

}

void _CYCLIC paiMpCyclic(void)
{
	paiMpComCyclic();

	paiMpFileManagerCyclic();

	paiMpRecipeCyclic();
	paiMpRecipeCustom1Cyclic();
	paiMpRecipeCustom2Cyclic();

	paiMpAlarmCyclic();

}
//EOF
```

### Program Logical/paiComponents/paiPing/paiPingService (ANSIC) - pai Ping Service (TK#8)

#### paiPingService.c
```c
/********************************************************************
 * COPYRIGHT --
 ********************************************************************
 * Program: paiPingService
 * File: paiPingService.c
 * Author: goran
 * Created: August 17, 2015
 ********************************************************************
 * Implementation of program paiPingService
 ********************************************************************/

#include <bur/plctypes.h>

#ifdef _DEFAULT_INCLUDES
	#include <AsDefault.h>
#endif

void paiPingInit(paiPing_typ* p, UDINT pingIntervalXms, UDINT pingTimeoutXms);
void paiPingCyclic(paiPing_typ* p);

void _INIT paiPingServiceInit(void)
{
	/* TODO: Add code here */
	brsstrcpy((UDINT)gPaiPing.iIPAddrStr, (UDINT)gPaiConfigSys.paiSys.ethernet.ipAddr);
	paiPingInit(&gPaiPing, 3000, 1000);
}

void _CYCLIC paiPingServiceCyclic(void)
{
	/* TODO: Add code here */
	paiPingCyclic(&gPaiPing);
}
```

### Package Logical/paiComponents/paiTemplate/paiHMI/paiScreens - Package

- lightFeature.clm (not shown)

- pageTabs.clm (not shown)

- pageTabsLines.clm (not shown)

- shiftStatus.clm (not shown)

- AlarmPopUp.fninfo (not shown)

- Arial14px.fninfo (not shown)

- Arial14pxBold.fninfo (not shown)

- Arial9pxValue.fninfo (not shown)

- CourierNew12px.fninfo (not shown)

- DateTime.fninfo (not shown)

- Default_0.fninfo (not shown)

- DefaultFont.fninfo (not shown)

- Html_SDM_0.fninfo (not shown)

- HugeText.fninfo (not shown)

- Info.fninfo (not shown)

- Info_0.fninfo (not shown)

- Info_1.fninfo (not shown)

- Input_0.fninfo (not shown)

- LargeText.fninfo (not shown)

- MenuItems.fninfo (not shown)

- MpDefault.fninfo (not shown)

- MpHeader.fninfo (not shown)

- MpHeader2.fninfo (not shown)

- MpHtml_SDM.fninfo (not shown)

- MpInput.fninfo (not shown)

- MpMenuButtons.fninfo (not shown)

- MpPackMLStateNames.fninfo (not shown)

- MpPads.fninfo (not shown)

- Pads.fninfo (not shown)

- Pads_0.fninfo (not shown)

- Status_0.fninfo (not shown)

- TabButtonTextSmall.fninfo (not shown)

- Background.layer (not shown)

- globalArea.layer (not shown)

- MpPageControl.layer (not shown)

- paiHmiTabs8.layer (not shown)

- paiHmiTabs9.layer (not shown)

- paiMpComLoggerUI.layer (not shown)

- EditPad2.tpr (not shown)

- NavigationPad_hor2.tpr (not shown)

- Trend_Temperature.tre (not shown)

### Program Logical/paiComponents/paiTemplate/paiHMI/paiHmi (ANSIC) - pai HMITemplate Support (TK#8) 

#### paiHmi.c - Implementation code
```c
/********************************************************************
 * COPYRIGHT --
 ********************************************************************
 * Program: paiHmi
 * File: paiHmi.c
 * Author: goran
 * Created: July 27, 2015
 ********************************************************************
 * Implementation of program paiHmi
 ********************************************************************/

#include <bur/plctypes.h>

#ifdef _DEFAULT_INCLUDES
	#include <AsDefault.h>
#endif

#include "../../../paiHmi/paiHmiParamList.h"
#include "../../../paiHmi/paiHmiDialog.h"
#include "../../../paiHmi/paiHmiAlert.h"
#include "../../../paiHmi/paiHmiSystemDateTime.h"
#include "../../../paiHmi/paiHmiSystemNetworking.h"
#include "../../../paiHmi/paiHmiMsgScrolling.h"
#include "../../../paiHmi/paiHmiLFMenuTabsPages.h"
#include "../../../paiHmi/paiHmiDropdownMenuRT.h"

/**
Recipe and config support cyclic logic. Monitors recipe and config changes (a change indication provided by recipe and config subsystem)
and controls visibility of the global buttons that allows user to trigger recipe and config save actions.
Prompts the user to make a decession about saving changes using an HMI dialog. Based on the user input,
it than notifies the recipe and config subsystem to either accept or discard changes in active recipe or config.
NOTE: uses global variables
*/
#if 0
static void recipeSaveCyclic()
{
	UINT ret;

	//control visibility: save cfg button
	//NOTE: button is not visible during setting of a new recipe! During that time, active recipe is in transition and it should not be
	//posible to store it
//	bgBitSetUINT(&gHmi.status.visibleSaveCfg, 0, (gConfig.out.isChanged)?0:1);

	//NOTE: visibility of this button is controlled! This action is only possible when the button is visible!
//	if(gHmi.keys.btnSaveCfg){
//		DBG(lgr, "save cfg request");
//		gHmi.keys.btnSaveCfg = 0;
		paiHmiDialogShow(&gPaiHmiDialogMsg, "Save Machine Config Changes?", 10000, 1, 2, 0);
//	}

	ret = paiHmiDialogCyclic(&gPaiHmiDialogMsg);
	if(ret == 1){
		//save config accepted
//		DBG(lgr, "save cfg accepted!");
		paiHmiAlertShow(&gPaiHmiAlertMsg, "Machine Config changes saved.", 2000);
//		gConfig.in.isChangeAccepted = 1;

	}
	if(ret == 2){
		//save config canceled
//		DBG(lgr, "save cfg rejected!");
		paiHmiAlertShow(&gPaiHmiAlertMsg, "Machine Config changes NOT saved.\nValues restored.", 3000);
//		gConfig.in.isChangeRejected = 1;
	}

	paiHmiAlertCyclic(&gPaiHmiAlertMsg);

}
#endif

void _INIT paiHmiInit(void)
{
	/* TODO: Add code here */

	//Message scrolling support - init
	gPaiHmiMsgScroll.iEnable = 1;
	paiHmiMsgScrollingInit(&gPaiHmiMsgScroll, (UDINT)&gAlarmsFiltered.alarmActive[0], APP_ALARM_LAST + 1, 3000);

	//Support for alert message - init
	paiHmiAlertHide(&gPaiHmiAlertMsg);

	//Support for dialog message - init
	paiHmiDialogHide(&gPaiHmiDialogMsg);

	//Support for RT drop-down menu
	gPaiHmiRTMenu.iMenuRTTimeout = 5.0;//gConfig.active.paiHmi.timerSettings.dropdwMenuRTTimeout;
	paiHmiDropDownMenuRTInit(&gPaiHmiRTMenu);

	//System Date & Time support
	paiHmiSystemDateTimeInit(&gPaiHmiSystemDateTime);

	//Screensaver support
	if(gScrensaverTimeout < 60){
		gScrensaverTimeout = 60;
	}

	/*
###############################################################################
	PAI_CONFIGURATION_SECTION
	Enter correct IF for the Ethernet port.
###############################################################################
	*/
	//System networking
	brsstrcpy((UDINT)gPaiConfigSys.paiSys.ethernet.ethDevice, (UDINT)"IF2");
	gPaiHmiNetworking.iPtrNWConfig = &gPaiConfigSys.paiSys.ethernet;
	paiHmiSystemNetworkingInit(&gPaiHmiNetworking);

}

void _CYCLIC paiHmiCyclic(void)
{
	/* TODO: Add code here */

	/*
###############################################################################
	PAI_CONFIGURATION_SECTION
	Code below allows configuration of VC resource used in this project.
	Enter correct name of the VC object.
###############################################################################
	*/
#warning "pai Configuration: HMI and Visual Components"

	//Page navigation using dropdown Menu (upper left corner) and Tabs
	paiHmiPageNavLFMenuTabsCyclic(&gPaiHmiMain, "WSVGA", 15);

	//Message scrolling support - cyclic
	paiHmiMsgScrollingCyclic(&gPaiHmiMsgScroll);

	//Support for RT drop-down menu
	paiHmiDropDownMenuRTCyclic(&gPaiHmiRTMenu);

	//System Date & Time support
	paiHmiSystemDateTimeCyclic(&gPaiHmiSystemDateTime);

	//System networking
	paiHmiSystemNetworkingCyclic(&gPaiHmiNetworking);

	//Alert cyclic control
	paiHmiAlertCyclic(&gPaiHmiAlertMsg);

	//Support for dialog message - cyclic
	paiHmiDialogCyclic(&gPaiHmiDialogMsg);

}
```

- bgstring.c (reference to Logical/paiComponents/bglib/bgstring.c)

- bgBitUtilities.c (reference to Logical/paiComponents/bglib/bgBitUtilities.c)

- paiHmiLFMenuTabsPages.c (reference to Logical/paiComponents/paiHmi/paiHmiLFMenuTabsPages.c)

- paiHmiMsgScrolling.c (reference to Logical/paiComponents/paiHmi/paiHmiMsgScrolling.c)

- paiHmiDropdownMenuRT.c (reference to Logical/paiComponents/paiHmi/paiHmiDropdownMenuRT.c)

- paiHmiSystemNetworking.c (reference to Logical/paiComponents/paiHmi/paiHmiSystemNetworking.c)

### udpApp.var
```iecst
(********************************************************************
 * COPYRIGHT -- HP
 ********************************************************************
 * File: Global.var
 * Author: goran
 * Created: January 23, 2013
 ********************************************************************
 * Global variables of project YieldPlus
 ********************************************************************)
VAR
	gUdpRxState : UDINT := 0;
	gUdpCommTimeoutTmr : TON := (0);
END_VAR
```
